    CONST robtarget Target_7240:=[[97.404735669,131.379041523,0],[0,0,1,0],[0,0,0,0],[9E+09,9E+09,9E+09,9E+09,9E+09,9E+09]];
    CONST robtarget Target_7250:=[[104.308059394,134.057322127,0],[0,0,1,0],[0,0,0,0],[9E+09,9E+09,9E+09,9E+09,9E+09,9E+09]];
    CONST robtarget Target_7260:=[[111.293699053,136.477383043,0],[0,0,1,0],[0,0,0,0],[9E+09,9E+09,9E+09,9E+09,9E+09,9E+09]];
    CONST robtarget Target_7270:=[[115.08379892,137.360119805,0],[0,0,1,0],[0,0,0,0],[9E+09,9E+09,9E+09,9E+09,9E+09,9E+09]];
    CONST robtarget Target_7280:=[[119.016514302,137.798137565,0],[0,0,1,0],[0,0,0,0],[9E+09,9E+09,9E+09,9E+09,9E+09,9E+09]];
    CONST robtarget Target_7290:=[[126.994438246,138.21544406,0],[0,0,1,0],[0,0,0,0],[9E+09,9E+09,9E+09,9E+09,9E+09,9E+09]];
    CONST robtarget Target_7300:=[[128.009308622,138.133836593,0],[0,0,1,0],[0,0,0,0],[9E+09,9E+09,9E+09,9E+09,9E+09,9E+09]];
    CONST robtarget Target_7310:=[[129.094775731,137.821862787,0],[0,0,1,0],[0,0,0,0],[9E+09,9E+09,9E+09,9E+09,9E+09,9E+09]];
    CONST robtarget Target_7320:=[[131.666016764,136.934701488,0],[0,0,1,0],[0,0,0,0],[9E+09,9E+09,9E+09,9E+09,9E+09,9E+09]];
    CONST robtarget Target_7330:=[[115.036980299,130.031874476,0],[0,0,1,0],[0,0,0,0],[9E+09,9E+09,9E+09,9E+09,9E+09,9E+09]];
    CONST robtarget Target_7330_2:=[[115.036980299,130.031874476,20],[0,0,1,0],[0,0,0,0],[9E+09,9E+09,9E+09,9E+09,9E+09,9E+09]];
    CONST robtarget Target_7340_2:=[[129.876572493,85.549987473,20],[0,0,1,0],[0,0,0,0],[9E+09,9E+09,9E+09,9E+09,9E+09,9E+09]];
    CONST robtarget Target_7340:=[[129.876572493,85.549987473,0],[0,0,1,0],[0,0,0,0],[9E+09,9E+09,9E+09,9E+09,9E+09,9E+09]];
    CONST robtarget Target_7350:=[[129.333218932,86.748318348,0],[0,0,1,0],[0,0,0,0],[9E+09,9E+09,9E+09,9E+09,9E+09,9E+09]];
    CONST robtarget Target_7360:=[[120.656332036,84.597871563,0],[0,0,1,0],[0,0,0,0],[9E+09,9E+09,9E+09,9E+09,9E+09,9E+09]];
    CONST robtarget Target_7370:=[[116.357422703,83.423068967,0],[0,0,1,0],[0,0,0,0],[9E+09,9E+09,9E+09,9E+09,9E+09,9E+09]];
    CONST robtarget Target_7380:=[[112.166530873,81.976192315,0],[0,0,1,0],[0,0,0,0],[9E+09,9E+09,9E+09,9E+09,9E+09,9E+09]];
    CONST robtarget Target_7390:=[[106.124575096,79.401977146,0],[0,0,1,0],[0,0,0,0],[9E+09,9E+09,9E+09,9E+09,9E+09,9E+09]];
    CONST robtarget Target_7400:=[[88.244330691,71.049330005,0],[0,0,1,0],[0,0,0,0],[9E+09,9E+09,9E+09,9E+09,9E+09,9E+09]];
    CONST robtarget Target_7410:=[[84.481212005,69.620753442,0],[0,0,1,0],[0,0,0,0],[9E+09,9E+09,9E+09,9E+09,9E+09,9E+09]];
    CONST robtarget Target_7420:=[[80.716429491,68.637006398,0],[0,0,1,0],[0,0,0,0],[9E+09,9E+09,9E+09,9E+09,9E+09,9E+09]];
    CONST robtarget Target_7430:=[[76.954340789,68.092878497,0],[0,0,1,0],[0,0,0,0],[9E+09,9E+09,9E+09,9E+09,9E+09,9E+09]];
    CONST robtarget Target_7440:=[[73.199303537,67.983159363,0],[0,0,1,0],[0,0,0,0],[9E+09,9E+09,9E+09,9E+09,9E+09,9E+09]];
    CONST robtarget Target_7450:=[[69.455675374,68.302638618,0],[0,0,1,0],[0,0,0,0],[9E+09,9E+09,9E+09,9E+09,9E+09,9E+09]];
    CONST robtarget Target_7460:=[[65.727813937,69.046105887,0],[0,0,1,0],[0,0,0,0],[9E+09,9E+09,9E+09,9E+09,9E+09,9E+09]];
    CONST robtarget Target_7470:=[[62.020076867,70.208350794,0],[0,0,1,0],[0,0,0,0],[9E+09,9E+09,9E+09,9E+09,9E+09,9E+09]];
    CONST robtarget Target_7480:=[[58.336821801,71.78416296,0],[0,0,1,0],[0,0,0,0],[9E+09,9E+09,9E+09,9E+09,9E+09,9E+09]];
    CONST robtarget Target_7490:=[[56.763326351,72.672328805,0],[0,0,1,0],[0,0,0,0],[9E+09,9E+09,9E+09,9E+09,9E+09,9E+09]];
    CONST robtarget Target_7500:=[[55.419669303,73.685478708,0],[0,0,1,0],[0,0,0,0],[9E+09,9E+09,9E+09,9E+09,9E+09,9E+09]];
    CONST robtarget Target_7510:=[[54.298199796,74.808495832,0],[0,0,1,0],[0,0,0,0],[9E+09,9E+09,9E+09,9E+09,9E+09,9E+09]];
    CONST robtarget Target_7520:=[[53.391266972,76.026263336,0],[0,0,1,0],[0,0,0,0],[9E+09,9E+09,9E+09,9E+09,9E+09,9E+09]];
    CONST robtarget Target_7530:=[[52.691219971,77.323664383,0],[0,0,1,0],[0,0,0,0],[9E+09,9E+09,9E+09,9E+09,9E+09,9E+09]];
    CONST robtarget Target_7540:=[[52.190407933,78.685582133,0],[0,0,1,0],[0,0,0,0],[9E+09,9E+09,9E+09,9E+09,9E+09,9E+09]];
    CONST robtarget Target_7550:=[[51.755885311,81.542500387,0],[0,0,1,0],[0,0,0,0],[9E+09,9E+09,9E+09,9E+09,9E+09,9E+09]];
    CONST robtarget Target_7560:=[[52.026492229,84.476083387,0],[0,0,1,0],[0,0,0,0],[9E+09,9E+09,9E+09,9E+09,9E+09,9E+09]];
    CONST robtarget Target_7570:=[[52.941021811,87.365396422,0],[0,0,1,0],[0,0,0,0],[9E+09,9E+09,9E+09,9E+09,9E+09,9E+09]];
    CONST robtarget Target_7580:=[[54.438267181,90.089504782,0],[0,0,1,0],[0,0,0,0],[9E+09,9E+09,9E+09,9E+09,9E+09,9E+09]];
    CONST robtarget Target_7590:=[[56.457021465,92.527473754,0],[0,0,1,0],[0,0,0,0],[9E+09,9E+09,9E+09,9E+09,9E+09,9E+09]];
    CONST robtarget Target_7600:=[[56.316335288,88.929115434,0],[0,0,1,0],[0,0,0,0],[9E+09,9E+09,9E+09,9E+09,9E+09,9E+09]];
    CONST robtarget Target_7610:=[[56.453523859,85.970317693,0],[0,0,1,0],[0,0,0,0],[9E+09,9E+09,9E+09,9E+09,9E+09,9E+09]];
    CONST robtarget Target_7620:=[[56.93899034,83.536042059,0],[0,0,1,0],[0,0,0,0],[9E+09,9E+09,9E+09,9E+09,9E+09,9E+09]];
    CONST robtarget Target_7630:=[[57.843137896,81.511250063,0],[0,0,1,0],[0,0,0,0],[9E+09,9E+09,9E+09,9E+09,9E+09,9E+09]];
    CONST robtarget Target_7640:=[[59.23636969,79.780903236,0],[0,0,1,0],[0,0,0,0],[9E+09,9E+09,9E+09,9E+09,9E+09,9E+09]];
    CONST robtarget Target_7650:=[[61.189088885,78.229963107,0],[0,0,1,0],[0,0,0,0],[9E+09,9E+09,9E+09,9E+09,9E+09,9E+09]];
    CONST robtarget Target_7660:=[[63.771698646,76.743391208,0],[0,0,1,0],[0,0,0,0],[9E+09,9E+09,9E+09,9E+09,9E+09,9E+09]];
    CONST robtarget Target_7670:=[[67.054602136,75.206149067,0],[0,0,1,0],[0,0,0,0],[9E+09,9E+09,9E+09,9E+09,9E+09,9E+09]];
    CONST robtarget Target_7680:=[[68.464100111,74.610784942,0],[0,0,1,0],[0,0,0,0],[9E+09,9E+09,9E+09,9E+09,9E+09,9E+09]];
    CONST robtarget Target_7690:=[[71.32349125,73.279802023,0],[0,0,1,0],[0,0,0,0],[9E+09,9E+09,9E+09,9E+09,9E+09,9E+09]];
    CONST robtarget Target_7700:=[[74.141087214,72.412520642,0],[0,0,1,0],[0,0,0,0],[9E+09,9E+09,9E+09,9E+09,9E+09,9E+09]];
    CONST robtarget Target_7710:=[[76.925445565,71.99176175,0],[0,0,1,0],[0,0,0,0],[9E+09,9E+09,9E+09,9E+09,9E+09,9E+09]];
    CONST robtarget Target_7720:=[[79.685123865,72.000346299,0],[0,0,1,0],[0,0,0,0],[9E+09,9E+09,9E+09,9E+09,9E+09,9E+09]];
    CONST robtarget Target_7730:=[[82.428679675,72.421095242,0],[0,0,1,0],[0,0,0,0],[9E+09,9E+09,9E+09,9E+09,9E+09,9E+09]];
    CONST robtarget Target_7740:=[[85.164670556,73.236829529,0],[0,0,1,0],[0,0,0,0],[9E+09,9E+09,9E+09,9E+09,9E+09,9E+09]];
    CONST robtarget Target_7750:=[[87.901654071,74.430370112,0],[0,0,1,0],[0,0,0,0],[9E+09,9E+09,9E+09,9E+09,9E+09,9E+09]];
    CONST robtarget Target_7760:=[[94.465610205,78.171040828,0],[0,0,1,0],[0,0,0,0],[9E+09,9E+09,9E+09,9E+09,9E+09,9E+09]];
    CONST robtarget Target_7770:=[[98.441342552,80.111743376,0],[0,0,1,0],[0,0,0,0],[9E+09,9E+09,9E+09,9E+09,9E+09,9E+09]];
    CONST robtarget Target_7780:=[[106.616652637,83.542913403,0],[0,0,1,0],[0,0,0,0],[9E+09,9E+09,9E+09,9E+09,9E+09,9E+09]];
    CONST robtarget Target_7790:=[[116.490797826,87.190723014,0],[0,0,1,0],[0,0,0,0],[9E+09,9E+09,9E+09,9E+09,9E+09,9E+09]];
    CONST robtarget Target_7800:=[[126.476326895,90.545417185,0],[0,0,1,0],[0,0,0,0],[9E+09,9E+09,9E+09,9E+09,9E+09,9E+09]];
    CONST robtarget Target_7810:=[[132.154721448,92.265104517,0],[0,0,1,0],[0,0,0,0],[9E+09,9E+09,9E+09,9E+09,9E+09,9E+09]];
    CONST robtarget Target_7820:=[[137.901994386,93.748799757,0],[0,0,1,0],[0,0,0,0],[9E+09,9E+09,9E+09,9E+09,9E+09,9E+09]];
    CONST robtarget Target_7830:=[[138.868681172,94.121198932,0],[0,0,1,0],[0,0,0,0],[9E+09,9E+09,9E+09,9E+09,9E+09,9E+09]];
    CONST robtarget Target_7840:=[[140.005403026,94.778288617,0],[0,0,1,0],[0,0,0,0],[9E+09,9E+09,9E+09,9E+09,9E+09,9E+09]];
    CONST robtarget Target_7850:=[[142.426589149,96.658715467,0],[0,0,1,0],[0,0,0,0],[9E+09,9E+09,9E+09,9E+09,9E+09,9E+09]];
    CONST robtarget Target_7860:=[[144.440827175,98.81443219,0],[0,0,1,0],[0,0,0,0],[9E+09,9E+09,9E+09,9E+09,9E+09,9E+09]];
    CONST robtarget Target_7870:=[[145.068863909,99.81563422,0],[0,0,1,0],[0,0,0,0],[9E+09,9E+09,9E+09,9E+09,9E+09,9E+09]];
    CONST robtarget Target_7880:=[[146.276657484,118.119049392,0],[0,0,1,0],[0,0,0,0],[9E+09,9E+09,9E+09,9E+09,9E+09,9E+09]];
    CONST robtarget Target_7890:=[[146.64526605,126.844242033,0],[0,0,1,0],[0,0,0,0],[9E+09,9E+09,9E+09,9E+09,9E+09,9E+09]];
    CONST robtarget Target_7900:=[[146.787973419,135.569206509,0],[0,0,1,0],[0,0,0,0],[9E+09,9E+09,9E+09,9E+09,9E+09,9E+09]];
    CONST robtarget Target_7910:=[[146.562475324,139.254038779,0],[0,0,1,0],[0,0,0,0],[9E+09,9E+09,9E+09,9E+09,9E+09,9E+09]];
    CONST robtarget Target_7920:=[[145.921246168,142.96350994,0],[0,0,1,0],[0,0,0,0],[9E+09,9E+09,9E+09,9E+09,9E+09,9E+09]];
    CONST robtarget Target_7930:=[[144.906271256,146.595460317,0],[0,0,1,0],[0,0,0,0],[9E+09,9E+09,9E+09,9E+09,9E+09,9E+09]];
    CONST robtarget Target_7940:=[[143.559535893,150.04773023,0],[0,0,1,0],[0,0,0,0],[9E+09,9E+09,9E+09,9E+09,9E+09,9E+09]];
    CONST robtarget Target_7950:=[[142.098362485,152.988920359,0],[0,0,1,0],[0,0,0,0],[9E+09,9E+09,9E+09,9E+09,9E+09,9E+09]];
    CONST robtarget Target_7960:=[[140.597343597,155.290040678,0],[0,0,1,0],[0,0,0,0],[9E+09,9E+09,9E+09,9E+09,9E+09,9E+09]];
    CONST robtarget Target_7970:=[[138.979884765,156.940428018,0],[0,0,1,0],[0,0,0,0],[9E+09,9E+09,9E+09,9E+09,9E+09,9E+09]];
    CONST robtarget Target_7980:=[[137.169391522,157.929419214,0],[0,0,1,0],[0,0,0,0],[9E+09,9E+09,9E+09,9E+09,9E+09,9E+09]];
    CONST robtarget Target_7990:=[[135.089269401,158.246351098,0],[0,0,1,0],[0,0,0,0],[9E+09,9E+09,9E+09,9E+09,9E+09,9E+09]];
    CONST robtarget Target_8000:=[[132.662923938,157.880560503,0],[0,0,1,0],[0,0,0,0],[9E+09,9E+09,9E+09,9E+09,9E+09,9E+09]];
    CONST robtarget Target_8010:=[[131.295981682,157.438312036,0],[0,0,1,0],[0,0,0,0],[9E+09,9E+09,9E+09,9E+09,9E+09,9E+09]];
    CONST robtarget Target_8020:=[[129.813760666,156.821384262,0],[0,0,1,0],[0,0,0,0],[9E+09,9E+09,9E+09,9E+09,9E+09,9E+09]];
    CONST robtarget Target_8030:=[[128.206686581,156.028444284,0],[0,0,1,0],[0,0,0,0],[9E+09,9E+09,9E+09,9E+09,9E+09,9E+09]];
    CONST robtarget Target_8040:=[[126.465185118,155.058159208,0],[0,0,1,0],[0,0,0,0],[9E+09,9E+09,9E+09,9E+09,9E+09,9E+09]];
    CONST robtarget Target_8050:=[[109.498646442,144.635036292,0],[0,0,1,0],[0,0,0,0],[9E+09,9E+09,9E+09,9E+09,9E+09,9E+09]];
    CONST robtarget Target_8060:=[[106.871095834,143.600815978,0],[0,0,1,0],[0,0,0,0],[9E+09,9E+09,9E+09,9E+09,9E+09,9E+09]];
    CONST robtarget Target_8070:=[[104.040074599,143.129604341,0],[0,0,1,0],[0,0,0,0],[9E+09,9E+09,9E+09,9E+09,9E+09,9E+09]];
    CONST robtarget Target_8080:=[[102.705166463,143.724153708,0],[0,0,1,0],[0,0,0,0],[9E+09,9E+09,9E+09,9E+09,9E+09,9E+09]];
    CONST robtarget Target_8090:=[[101.793162077,144.941800307,0],[0,0,1,0],[0,0,0,0],[9E+09,9E+09,9E+09,9E+09,9E+09,9E+09]];
    CONST robtarget Target_8100:=[[101.495618729,147.367025782,0],[0,0,1,0],[0,0,0,0],[9E+09,9E+09,9E+09,9E+09,9E+09,9E+09]];
    CONST robtarget Target_8110:=[[101.657829955,149.725149825,0],[0,0,1,0],[0,0,0,0],[9E+09,9E+09,9E+09,9E+09,9E+09,9E+09]];
    CONST robtarget Target_8120:=[[102.392934157,151.976800956,0],[0,0,1,0],[0,0,0,0],[9E+09,9E+09,9E+09,9E+09,9E+09,9E+09]];
    CONST robtarget Target_8130:=[[103.814069741,154.082607694,0],[0,0,1,0],[0,0,0,0],[9E+09,9E+09,9E+09,9E+09,9E+09,9E+09]];
    CONST robtarget Target_8140:=[[105.014427772,152.941872808,0],[0,0,1,0],[0,0,0,0],[9E+09,9E+09,9E+09,9E+09,9E+09,9E+09]];
    CONST robtarget Target_8150:=[[106.090948335,152.075840773,0],[0,0,1,0],[0,0,0,0],[9E+09,9E+09,9E+09,9E+09,9E+09,9E+09]];
    CONST robtarget Target_8160:=[[107.094496065,151.472364639,0],[0,0,1,0],[0,0,0,0],[9E+09,9E+09,9E+09,9E+09,9E+09,9E+09]];
    CONST robtarget Target_8170:=[[108.075935597,151.11929746,0],[0,0,1,0],[0,0,0,0],[9E+09,9E+09,9E+09,9E+09,9E+09,9E+09]];
    CONST robtarget Target_8180:=[[109.086131569,151.004492288,0],[0,0,1,0],[0,0,0,0],[9E+09,9E+09,9E+09,9E+09,9E+09,9E+09]];
    CONST robtarget Target_8190:=[[110.175948615,151.115802173,0],[0,0,1,0],[0,0,0,0],[9E+09,9E+09,9E+09,9E+09,9E+09,9E+09]];
    CONST robtarget Target_8200:=[[111.396251371,151.441080169,0],[0,0,1,0],[0,0,0,0],[9E+09,9E+09,9E+09,9E+09,9E+09,9E+09]];
    CONST robtarget Target_8210:=[[112.797904472,151.968179326,0],[0,0,1,0],[0,0,0,0],[9E+09,9E+09,9E+09,9E+09,9E+09,9E+09]];
    CONST robtarget Target_8220:=[[115.564679196,153.274276463,0],[0,0,1,0],[0,0,0,0],[9E+09,9E+09,9E+09,9E+09,9E+09,9E+09]];
    CONST robtarget Target_8230:=[[132.009061776,159.756169017,0],[0,0,1,0],[0,0,0,0],[9E+09,9E+09,9E+09,9E+09,9E+09,9E+09]];
    CONST robtarget Target_8240:=[[134.035319183,160.214476419,0],[0,0,1,0],[0,0,0,0],[9E+09,9E+09,9E+09,9E+09,9E+09,9E+09]];
    CONST robtarget Target_8250:=[[135.93027141,160.027374554,0],[0,0,1,0],[0,0,0,0],[9E+09,9E+09,9E+09,9E+09,9E+09,9E+09]];
    CONST robtarget Target_8260:=[[137.707220601,159.295275159,0],[0,0,1,0],[0,0,0,0],[9E+09,9E+09,9E+09,9E+09,9E+09,9E+09]];
    CONST robtarget Target_8270:=[[139.379468904,158.118589974,0],[0,0,1,0],[0,0,0,0],[9E+09,9E+09,9E+09,9E+09,9E+09,9E+09]];
    CONST robtarget Target_8280:=[[142.735905784,155.157330385,0],[0,0,1,0],[0,0,0,0],[9E+09,9E+09,9E+09,9E+09,9E+09,9E+09]];
    CONST robtarget Target_8290:=[[146.248814226,158.507504441,0],[0,0,1,0],[0,0,0,0],[9E+09,9E+09,9E+09,9E+09,9E+09,9E+09]];
    CONST robtarget Target_8300:=[[149.181567375,162.145043518,0],[0,0,1,0],[0,0,0,0],[9E+09,9E+09,9E+09,9E+09,9E+09,9E+09]];
    CONST robtarget Target_8310:=[[151.588027369,166.046590479,0],[0,0,1,0],[0,0,0,0],[9E+09,9E+09,9E+09,9E+09,9E+09,9E+09]];
    CONST robtarget Target_8320:=[[153.522056348,170.188788191,0],[0,0,1,0],[0,0,0,0],[9E+09,9E+09,9E+09,9E+09,9E+09,9E+09]];
    CONST robtarget Target_8330:=[[155.037516447,174.548279518,0],[0,0,1,0],[0,0,0,0],[9E+09,9E+09,9E+09,9E+09,9E+09,9E+09]];
    CONST robtarget Target_8340:=[[156.188269805,179.101707326,0],[0,0,1,0],[0,0,0,0],[9E+09,9E+09,9E+09,9E+09,9E+09,9E+09]];
    CONST robtarget Target_8350:=[[157.02817856,183.82571448,0],[0,0,1,0],[0,0,0,0],[9E+09,9E+09,9E+09,9E+09,9E+09,9E+09]];
    CONST robtarget Target_8360:=[[157.61110485,188.696943846,0],[0,0,1,0],[0,0,0,0],[9E+09,9E+09,9E+09,9E+09,9E+09,9E+09]];
    CONST robtarget Target_8370:=[[159.511653012,185.615301707,0],[0,0,1,0],[0,0,0,0],[9E+09,9E+09,9E+09,9E+09,9E+09,9E+09]];
    CONST robtarget Target_8380:=[[160.122702203,184.061896932,0],[0,0,1,0],[0,0,0,0],[9E+09,9E+09,9E+09,9E+09,9E+09,9E+09]];
    CONST robtarget Target_8390:=[[160.269289382,182.540597159,0],[0,0,1,0],[0,0,0,0],[9E+09,9E+09,9E+09,9E+09,9E+09,9E+09]];
    CONST robtarget Target_8400:=[[159.048038496,172.743082596,0],[0,0,1,0],[0,0,0,0],[9E+09,9E+09,9E+09,9E+09,9E+09,9E+09]];
    CONST robtarget Target_8410:=[[157.272759984,163.030465722,0],[0,0,1,0],[0,0,0,0],[9E+09,9E+09,9E+09,9E+09,9E+09,9E+09]];
    CONST robtarget Target_8420:=[[152.804879363,147.17888185,0],[0,0,1,0],[0,0,0,0],[9E+09,9E+09,9E+09,9E+09,9E+09,9E+09]];
    CONST robtarget Target_8430:=[[152.522164651,144.959220559,0],[0,0,1,0],[0,0,0,0],[9E+09,9E+09,9E+09,9E+09,9E+09,9E+09]];
    CONST robtarget Target_8440:=[[152.513150484,142.629190929,0],[0,0,1,0],[0,0,0,0],[9E+09,9E+09,9E+09,9E+09,9E+09,9E+09]];
    CONST robtarget Target_8450:=[[152.692927912,137.569820222,0],[0,0,1,0],[0,0,0,0],[9E+09,9E+09,9E+09,9E+09,9E+09,9E+09]];
    CONST robtarget Target_8460:=[[156.030442498,141.602150995,0],[0,0,1,0],[0,0,0,0],[9E+09,9E+09,9E+09,9E+09,9E+09,9E+09]];
    CONST robtarget Target_8470:=[[156.030442498,132.222722326,0],[0,0,1,0],[0,0,0,0],[9E+09,9E+09,9E+09,9E+09,9E+09,9E+09]];
    CONST robtarget Target_8480:=[[157.683142524,134.267528632,0],[0,0,1,0],[0,0,0,0],[9E+09,9E+09,9E+09,9E+09,9E+09,9E+09]];
    CONST robtarget Target_8490:=[[158.819369695,133.854983277,0],[0,0,1,0],[0,0,0,0],[9E+09,9E+09,9E+09,9E+09,9E+09,9E+09]];
    CONST robtarget Target_8500:=[[162.027841116,110.98600871,0],[0,0,1,0],[0,0,0,0],[9E+09,9E+09,9E+09,9E+09,9E+09,9E+09]];
    CONST robtarget Target_8510:=[[181.059601621,117.520426784,0],[0,0,1,0],[0,0,0,0],[9E+09,9E+09,9E+09,9E+09,9E+09,9E+09]];
    CONST robtarget Target_8520:=[[182.051540866,118.158620642,0],[0,0,1,0],[0,0,0,0],[9E+09,9E+09,9E+09,9E+09,9E+09,9E+09]];
    CONST robtarget Target_8530:=[[182.911149594,119.054153231,0],[0,0,1,0],[0,0,0,0],[9E+09,9E+09,9E+09,9E+09,9E+09,9E+09]];
    CONST robtarget Target_8540:=[[185.369337847,121.989158564,0],[0,0,1,0],[0,0,0,0],[9E+09,9E+09,9E+09,9E+09,9E+09,9E+09]];
    CONST robtarget Target_8550:=[[187.52283735,125.030421014,0],[0,0,1,0],[0,0,0,0],[9E+09,9E+09,9E+09,9E+09,9E+09,9E+09]];
    CONST robtarget Target_8560:=[[189.341962726,128.188894081,0],[0,0,1,0],[0,0,0,0],[9E+09,9E+09,9E+09,9E+09,9E+09,9E+09]];
    CONST robtarget Target_8570:=[[190.797028597,131.475531266,0],[0,0,1,0],[0,0,0,0],[9E+09,9E+09,9E+09,9E+09,9E+09,9E+09]];
    CONST robtarget Target_8580:=[[191.858349584,134.90128607,0],[0,0,1,0],[0,0,0,0],[9E+09,9E+09,9E+09,9E+09,9E+09,9E+09]];
    CONST robtarget Target_8590:=[[192.496240311,138.477111994,0],[0,0,1,0],[0,0,0,0],[9E+09,9E+09,9E+09,9E+09,9E+09,9E+09]];
    CONST robtarget Target_8600:=[[192.6810154,142.213962539,0],[0,0,1,0],[0,0,0,0],[9E+09,9E+09,9E+09,9E+09,9E+09,9E+09]];
    CONST robtarget Target_8610:=[[192.382989472,146.122791206,0],[0,0,1,0],[0,0,0,0],[9E+09,9E+09,9E+09,9E+09,9E+09,9E+09]];
    CONST robtarget Target_8620:=[[192.420926442,148.208812875,0],[0,0,1,0],[0,0,0,0],[9E+09,9E+09,9E+09,9E+09,9E+09,9E+09]];
    CONST robtarget Target_8630:=[[192.684959714,150.325900139,0],[0,0,1,0],[0,0,0,0],[9E+09,9E+09,9E+09,9E+09,9E+09,9E+09]];
    CONST robtarget Target_8640:=[[194.072232654,150.218826726,0],[0,0,1,0],[0,0,0,0],[9E+09,9E+09,9E+09,9E+09,9E+09,9E+09]];
    CONST robtarget Target_8650:=[[195.747139356,143.338811976,0],[0,0,1,0],[0,0,0,0],[9E+09,9E+09,9E+09,9E+09,9E+09,9E+09]];
    CONST robtarget Target_8660:=[[196.664125368,136.503126165,0],[0,0,1,0],[0,0,0,0],[9E+09,9E+09,9E+09,9E+09,9E+09,9E+09]];
    CONST robtarget Target_8670:=[[196.884999904,129.708154654,0],[0,0,1,0],[0,0,0,0],[9E+09,9E+09,9E+09,9E+09,9E+09,9E+09]];
    CONST robtarget Target_8680:=[[196.471572174,122.950282803,0],[0,0,1,0],[0,0,0,0],[9E+09,9E+09,9E+09,9E+09,9E+09,9E+09]];
    CONST robtarget Target_8690:=[[195.485651391,116.22589597,0],[0,0,1,0],[0,0,0,0],[9E+09,9E+09,9E+09,9E+09,9E+09,9E+09]];
    CONST robtarget Target_8700:=[[193.989046766,109.531379516,0],[0,0,1,0],[0,0,0,0],[9E+09,9E+09,9E+09,9E+09,9E+09,9E+09]];
    CONST robtarget Target_8710:=[[192.043567513,102.863118799,0],[0,0,1,0],[0,0,0,0],[9E+09,9E+09,9E+09,9E+09,9E+09,9E+09]];
    CONST robtarget Target_8720:=[[189.711022843,96.217499179,0],[0,0,1,0],[0,0,0,0],[9E+09,9E+09,9E+09,9E+09,9E+09,9E+09]];
    CONST robtarget Target_8730:=[[196.507207134,106.638206483,0],[0,0,1,0],[0,0,0,0],[9E+09,9E+09,9E+09,9E+09,9E+09,9E+09]];
    CONST robtarget Target_8740:=[[194.822794884,94.14058975,0],[0,0,1,0],[0,0,0,0],[9E+09,9E+09,9E+09,9E+09,9E+09,9E+09]];
    CONST robtarget Target_8750:=[[191.767984454,82.136505163,0],[0,0,1,0],[0,0,0,0],[9E+09,9E+09,9E+09,9E+09,9E+09,9E+09]];
    CONST robtarget Target_8760:=[[188.283605859,70.215200936,0],[0,0,1,0],[0,0,0,0],[9E+09,9E+09,9E+09,9E+09,9E+09,9E+09]];
    CONST robtarget Target_8770:=[[184.439576675,58.342610969,0],[0,0,1,0],[0,0,0,0],[9E+09,9E+09,9E+09,9E+09,9E+09,9E+09]];
    CONST robtarget Target_8780:=[[191.596791989,64.817986988,0],[0,0,1,0],[0,0,0,0],[9E+09,9E+09,9E+09,9E+09,9E+09,9E+09]];
    CONST robtarget Target_8790:=[[192.600244759,63.94724308,0],[0,0,1,0],[0,0,0,0],[9E+09,9E+09,9E+09,9E+09,9E+09,9E+09]];
    CONST robtarget Target_8800:=[[181.316386808,45.55735645,0],[0,0,1,0],[0,0,0,0],[9E+09,9E+09,9E+09,9E+09,9E+09,9E+09]];
    CONST robtarget Target_8810:=[[180.372261691,43.421039482,0],[0,0,1,0],[0,0,0,0],[9E+09,9E+09,9E+09,9E+09,9E+09,9E+09]];
    CONST robtarget Target_8820:=[[180.129144821,42.280955318,0],[0,0,1,0],[0,0,0,0],[9E+09,9E+09,9E+09,9E+09,9E+09,9E+09]];
    CONST robtarget Target_8830:=[[180.119797422,41.18562281,0],[0,0,1,0],[0,0,0,0],[9E+09,9E+09,9E+09,9E+09,9E+09,9E+09]];
    CONST robtarget Target_8840:=[[180.601400728,38.257669681,0],[0,0,1,0],[0,0,0,0],[9E+09,9E+09,9E+09,9E+09,9E+09,9E+09]];
    CONST robtarget Target_8850:=[[181.314808838,35.434360847,0],[0,0,1,0],[0,0,0,0],[9E+09,9E+09,9E+09,9E+09,9E+09,9E+09]];
    CONST robtarget Target_8860:=[[182.251851673,32.713303093,0],[0,0,1,0],[0,0,0,0],[9E+09,9E+09,9E+09,9E+09,9E+09,9E+09]];
    CONST robtarget Target_8870:=[[183.404359151,30.092103202,0],[0,0,1,0],[0,0,0,0],[9E+09,9E+09,9E+09,9E+09,9E+09,9E+09]];
    CONST robtarget Target_8880:=[[184.764161193,27.56836796,0],[0,0,1,0],[0,0,0,0],[9E+09,9E+09,9E+09,9E+09,9E+09,9E+09]];
    CONST robtarget Target_8890:=[[186.323087717,25.13970415,0],[0,0,1,0],[0,0,0,0],[9E+09,9E+09,9E+09,9E+09,9E+09,9E+09]];
    CONST robtarget Target_8900:=[[188.072968645,22.803718557,0],[0,0,1,0],[0,0,0,0],[9E+09,9E+09,9E+09,9E+09,9E+09,9E+09]];
    CONST robtarget Target_8910:=[[190.005633895,20.558017965,0],[0,0,1,0],[0,0,0,0],[9E+09,9E+09,9E+09,9E+09,9E+09,9E+09]];
    CONST robtarget Target_8920:=[[192.020885573,18.577072276,0],[0,0,1,0],[0,0,0,0],[9E+09,9E+09,9E+09,9E+09,9E+09,9E+09]];
    CONST robtarget Target_8930:=[[194.22441566,16.936248541,0],[0,0,1,0],[0,0,0,0],[9E+09,9E+09,9E+09,9E+09,9E+09,9E+09]];
    CONST robtarget Target_8940:=[[196.702778083,15.717678967,0],[0,0,1,0],[0,0,0,0],[9E+09,9E+09,9E+09,9E+09,9E+09,9E+09]];
    CONST robtarget Target_8950:=[[199.542526769,15.003495761,0],[0,0,1,0],[0,0,0,0],[9E+09,9E+09,9E+09,9E+09,9E+09,9E+09]];
    CONST robtarget Target_8960:=[[201.153882275,14.877956022,0],[0,0,1,0],[0,0,0,0],[9E+09,9E+09,9E+09,9E+09,9E+09,9E+09]];
    CONST robtarget Target_8970:=[[202.564135721,14.991268303,0],[0,0,1,0],[0,0,0,0],[9E+09,9E+09,9E+09,9E+09,9E+09,9E+09]];
    CONST robtarget Target_8980:=[[203.767899383,15.347108916,0],[0,0,1,0],[0,0,0,0],[9E+09,9E+09,9E+09,9E+09,9E+09,9E+09]];
    CONST robtarget Target_8990:=[[204.759785534,15.949154177,0],[0,0,1,0],[0,0,0,0],[9E+09,9E+09,9E+09,9E+09,9E+09,9E+09]];
    CONST robtarget Target_9000:=[[205.534406448,16.801080396,0],[0,0,1,0],[0,0,0,0],[9E+09,9E+09,9E+09,9E+09,9E+09,9E+09]];
    CONST robtarget Target_9010:=[[206.086374398,17.906563889,0],[0,0,1,0],[0,0,0,0],[9E+09,9E+09,9E+09,9E+09,9E+09,9E+09]];
    CONST robtarget Target_9020:=[[206.41030166,19.269280967,0],[0,0,1,0],[0,0,0,0],[9E+09,9E+09,9E+09,9E+09,9E+09,9E+09]];
    CONST robtarget Target_9030:=[[206.500800507,20.892907944,0],[0,0,1,0],[0,0,0,0],[9E+09,9E+09,9E+09,9E+09,9E+09,9E+09]];
    CONST robtarget Target_9040:=[[206.185218881,23.076640763,0],[0,0,1,0],[0,0,0,0],[9E+09,9E+09,9E+09,9E+09,9E+09,9E+09]];
    CONST robtarget Target_9050:=[[205.382591695,24.995387031,0],[0,0,1,0],[0,0,0,0],[9E+09,9E+09,9E+09,9E+09,9E+09,9E+09]];
    CONST robtarget Target_9060:=[[204.197106581,26.718523927,0],[0,0,1,0],[0,0,0,0],[9E+09,9E+09,9E+09,9E+09,9E+09,9E+09]];
    CONST robtarget Target_9070:=[[202.732951174,28.315428627,0],[0,0,1,0],[0,0,0,0],[9E+09,9E+09,9E+09,9E+09,9E+09,9E+09]];
    CONST robtarget Target_9080:=[[201.23516049,29.821989131,0],[0,0,1,0],[0,0,0,0],[9E+09,9E+09,9E+09,9E+09,9E+09,9E+09]];
    CONST robtarget Target_9090:=[[199.891820974,31.444879405,0],[0,0,1,0],[0,0,0,0],[9E+09,9E+09,9E+09,9E+09,9E+09,9E+09]];
    CONST robtarget Target_9100:=[[198.917384536,33.31544624,0],[0,0,1,0],[0,0,0,0],[9E+09,9E+09,9E+09,9E+09,9E+09,9E+09]];
    CONST robtarget Target_9110:=[[198.635521194,34.384654239,0],[0,0,1,0],[0,0,0,0],[9E+09,9E+09,9E+09,9E+09,9E+09,9E+09]];
    CONST robtarget Target_9120:=[[198.526303089,35.565036423,0],[0,0,1,0],[0,0,0,0],[9E+09,9E+09,9E+09,9E+09,9E+09,9E+09]];
    CONST robtarget Target_9130:=[[200.025047194,34.332688531,0],[0,0,1,0],[0,0,0,0],[9E+09,9E+09,9E+09,9E+09,9E+09,9E+09]];
    CONST robtarget Target_9140:=[[201.408478298,33.350226146,0],[0,0,1,0],[0,0,0,0],[9E+09,9E+09,9E+09,9E+09,9E+09,9E+09]];
    CONST robtarget Target_9150:=[[202.710907397,32.605760367,0],[0,0,1,0],[0,0,0,0],[9E+09,9E+09,9E+09,9E+09,9E+09,9E+09]];
    CONST robtarget Target_9160:=[[203.966645486,32.08740229,0],[0,0,1,0],[0,0,0,0],[9E+09,9E+09,9E+09,9E+09,9E+09,9E+09]];
    CONST robtarget Target_9170:=[[205.210003564,31.783263015,0],[0,0,1,0],[0,0,0,0],[9E+09,9E+09,9E+09,9E+09,9E+09,9E+09]];
    CONST robtarget Target_9180:=[[206.475292626,31.681453639,0],[0,0,1,0],[0,0,0,0],[9E+09,9E+09,9E+09,9E+09,9E+09,9E+09]];
    CONST robtarget Target_9190:=[[207.796823668,31.77008526,0],[0,0,1,0],[0,0,0,0],[9E+09,9E+09,9E+09,9E+09,9E+09,9E+09]];
    CONST robtarget Target_9200:=[[209.208907689,32.037268976,0],[0,0,1,0],[0,0,0,0],[9E+09,9E+09,9E+09,9E+09,9E+09,9E+09]];
    CONST robtarget Target_9210:=[[206.498192883,34.63263406,0],[0,0,1,0],[0,0,0,0],[9E+09,9E+09,9E+09,9E+09,9E+09,9E+09]];
    CONST robtarget Target_9220:=[[204.288706623,36.849937851,0],[0,0,1,0],[0,0,0,0],[9E+09,9E+09,9E+09,9E+09,9E+09,9E+09]];
    CONST robtarget Target_9230:=[[202.519543794,38.803163097,0],[0,0,1,0],[0,0,0,0],[9E+09,9E+09,9E+09,9E+09,9E+09,9E+09]];
    CONST robtarget Target_9240:=[[201.129799285,40.606292545,0],[0,0,1,0],[0,0,0,0],[9E+09,9E+09,9E+09,9E+09,9E+09,9E+09]];
    CONST robtarget Target_9250:=[[200.058567982,42.373308942,0],[0,0,1,0],[0,0,0,0],[9E+09,9E+09,9E+09,9E+09,9E+09,9E+09]];
    CONST robtarget Target_9260:=[[199.244944772,44.218195037,0],[0,0,1,0],[0,0,0,0],[9E+09,9E+09,9E+09,9E+09,9E+09,9E+09]];
    CONST robtarget Target_9270:=[[198.628024542,46.254933577,0],[0,0,1,0],[0,0,0,0],[9E+09,9E+09,9E+09,9E+09,9E+09,9E+09]];
    CONST robtarget Target_9280:=[[198.146902179,48.597507309,0],[0,0,1,0],[0,0,0,0],[9E+09,9E+09,9E+09,9E+09,9E+09,9E+09]];
    CONST robtarget Target_9290:=[[196.61288422,59.686081257,0],[0,0,1,0],[0,0,0,0],[9E+09,9E+09,9E+09,9E+09,9E+09,9E+09]];
    CONST robtarget Target_9300:=[[196.174396262,65.230484615,0],[0,0,1,0],[0,0,0,0],[9E+09,9E+09,9E+09,9E+09,9E+09,9E+09]];
    CONST robtarget Target_9310:=[[196.004662814,70.774974464,0],[0,0,1,0],[0,0,0,0],[9E+09,9E+09,9E+09,9E+09,9E+09,9E+09]];
    CONST robtarget Target_9320:=[[196.140989249,76.31955748,0],[0,0,1,0],[0,0,0,0],[9E+09,9E+09,9E+09,9E+09,9E+09,9E+09]];
    CONST robtarget Target_9330:=[[196.620680938,81.864240338,0],[0,0,1,0],[0,0,0,0],[9E+09,9E+09,9E+09,9E+09,9E+09,9E+09]];
    CONST robtarget Target_9340:=[[197.481043255,87.409029715,0],[0,0,1,0],[0,0,0,0],[9E+09,9E+09,9E+09,9E+09,9E+09,9E+09]];
    CONST robtarget Target_9350:=[[198.759381571,92.953932286,0],[0,0,1,0],[0,0,0,0],[9E+09,9E+09,9E+09,9E+09,9E+09,9E+09]];
    CONST robtarget Target_9360:=[[201.564466199,104.252177175,0],[0,0,1,0],[0,0,0,0],[9E+09,9E+09,9E+09,9E+09,9E+09,9E+09]];
    CONST robtarget Target_9370:=[[203.789655734,115.652677805,0],[0,0,1,0],[0,0,0,0],[9E+09,9E+09,9E+09,9E+09,9E+09,9E+09]];
    CONST robtarget Target_9380:=[[204.636408963,121.396078998,0],[0,0,1,0],[0,0,0,0],[9E+09,9E+09,9E+09,9E+09,9E+09,9E+09]];
    CONST robtarget Target_9390:=[[205.280131364,127.170810095,0],[0,0,1,0],[0,0,0,0],[9E+09,9E+09,9E+09,9E+09,9E+09,9E+09]];
    CONST robtarget Target_9400:=[[205.701470586,132.978793087,0],[0,0,1,0],[0,0,0,0],[9E+09,9E+09,9E+09,9E+09,9E+09,9E+09]];
    CONST robtarget Target_9410:=[[205.881074278,138.821949962,0],[0,0,1,0],[0,0,0,0],[9E+09,9E+09,9E+09,9E+09,9E+09,9E+09]];
    CONST robtarget Target_9420:=[[205.923787544,163.023012903,0],[0,0,1,0],[0,0,0,0],[9E+09,9E+09,9E+09,9E+09,9E+09,9E+09]];
    CONST robtarget Target_9430:=[[206.224124409,164.437566789,0],[0,0,1,0],[0,0,0,0],[9E+09,9E+09,9E+09,9E+09,9E+09,9E+09]];
    CONST robtarget Target_9440:=[[206.729796792,165.850533718,0],[0,0,1,0],[0,0,0,0],[9E+09,9E+09,9E+09,9E+09,9E+09,9E+09]];
    CONST robtarget Target_9450:=[[207.958631791,165.588804952,0],[0,0,1,0],[0,0,0,0],[9E+09,9E+09,9E+09,9E+09,9E+09,9E+09]];
    CONST robtarget Target_9460:=[[207.958631791,150.141115173,0],[0,0,1,0],[0,0,0,0],[9E+09,9E+09,9E+09,9E+09,9E+09,9E+09]];
    CONST robtarget Target_9470:=[[209.430226624,151.721456097,0],[0,0,1,0],[0,0,0,0],[9E+09,9E+09,9E+09,9E+09,9E+09,9E+09]];
    CONST robtarget Target_9480:=[[210.695447211,153.379474728,0],[0,0,1,0],[0,0,0,0],[9E+09,9E+09,9E+09,9E+09,9E+09,9E+09]];
    CONST robtarget Target_9490:=[[211.761289196,155.107679103,0],[0,0,1,0],[0,0,0,0],[9E+09,9E+09,9E+09,9E+09,9E+09,9E+09]];
    CONST robtarget Target_9500:=[[212.634748223,156.898577253,0],[0,0,1,0],[0,0,0,0],[9E+09,9E+09,9E+09,9E+09,9E+09,9E+09]];
    CONST robtarget Target_9510:=[[213.832499974,160.638487019,0],[0,0,1,0],[0,0,0,0],[9E+09,9E+09,9E+09,9E+09,9E+09,9E+09]];
    CONST robtarget Target_9520:=[[214.344667613,164.539268295,0],[0,0,1,0],[0,0,0,0],[9E+09,9E+09,9E+09,9E+09,9E+09,9E+09]];
    CONST robtarget Target_9530:=[[215.042181606,177.509334354,0],[0,0,1,0],[0,0,0,0],[9E+09,9E+09,9E+09,9E+09,9E+09,9E+09]];
    CONST robtarget Target_9540:=[[215.288779154,183.99202098,0],[0,0,1,0],[0,0,0,0],[9E+09,9E+09,9E+09,9E+09,9E+09,9E+09]];
    CONST robtarget Target_9550:=[[215.321559695,190.464065247,0],[0,0,1,0],[0,0,0,0],[9E+09,9E+09,9E+09,9E+09,9E+09,9E+09]];
    CONST robtarget Target_9560:=[[215.0312402,196.918658587,0],[0,0,1,0],[0,0,0,0],[9E+09,9E+09,9E+09,9E+09,9E+09,9E+09]];
    CONST robtarget Target_9570:=[[214.308537638,203.348992435,0],[0,0,1,0],[0,0,0,0],[9E+09,9E+09,9E+09,9E+09,9E+09,9E+09]];
    CONST robtarget Target_9580:=[[213.044168979,209.748258222,0],[0,0,1,0],[0,0,0,0],[9E+09,9E+09,9E+09,9E+09,9E+09,9E+09]];
    CONST robtarget Target_9590:=[[211.128851192,216.109647382,0],[0,0,1,0],[0,0,0,0],[9E+09,9E+09,9E+09,9E+09,9E+09,9E+09]];
    CONST robtarget Target_9600:=[[210.788553003,217.797412552,0],[0,0,1,0],[0,0,0,0],[9E+09,9E+09,9E+09,9E+09,9E+09,9E+09]];
    CONST robtarget Target_9610:=[[210.788455864,219.607370654,0],[0,0,1,0],[0,0,0,0],[9E+09,9E+09,9E+09,9E+09,9E+09,9E+09]];
    CONST robtarget Target_9620:=[[211.023875056,223.31191667,0],[0,0,1,0],[0,0,0,0],[9E+09,9E+09,9E+09,9E+09,9E+09,9E+09]];
    CONST robtarget Target_9630:=[[212.166253612,223.389478418,0],[0,0,1,0],[0,0,0,0],[9E+09,9E+09,9E+09,9E+09,9E+09,9E+09]];
    CONST robtarget Target_9640:=[[214.81517292,218.24211088,0],[0,0,1,0],[0,0,0,0],[9E+09,9E+09,9E+09,9E+09,9E+09,9E+09]];
    CONST robtarget Target_9650:=[[216.899235082,212.99446713,0],[0,0,1,0],[0,0,0,0],[9E+09,9E+09,9E+09,9E+09,9E+09,9E+09]];
    CONST robtarget Target_9660:=[[218.451485575,207.65318286,0],[0,0,1,0],[0,0,0,0],[9E+09,9E+09,9E+09,9E+09,9E+09,9E+09]];
    CONST robtarget Target_9670:=[[219.504969875,202.224893763,0],[0,0,1,0],[0,0,0,0],[9E+09,9E+09,9E+09,9E+09,9E+09,9E+09]];
    CONST robtarget Target_9680:=[[220.09273346,196.71623553,0],[0,0,1,0],[0,0,0,0],[9E+09,9E+09,9E+09,9E+09,9E+09,9E+09]];
    CONST robtarget Target_9690:=[[220.247821808,191.133843852,0],[0,0,1,0],[0,0,0,0],[9E+09,9E+09,9E+09,9E+09,9E+09,9E+09]];
    CONST robtarget Target_9700:=[[220.003280397,185.484354422,0],[0,0,1,0],[0,0,0,0],[9E+09,9E+09,9E+09,9E+09,9E+09,9E+09]];
    CONST robtarget Target_9710:=[[219.392154702,179.774402932,0],[0,0,1,0],[0,0,0,0],[9E+09,9E+09,9E+09,9E+09,9E+09,9E+09]];
    CONST robtarget Target_9720:=[[222.818953308,182.875955281,0],[0,0,1,0],[0,0,0,0],[9E+09,9E+09,9E+09,9E+09,9E+09,9E+09]];
    CONST robtarget Target_9730:=[[221.216466181,170.263445118,0],[0,0,1,0],[0,0,0,0],[9E+09,9E+09,9E+09,9E+09,9E+09,9E+09]];
    CONST robtarget Target_9740:=[[224.690584569,174.489773888,0],[0,0,1,0],[0,0,0,0],[9E+09,9E+09,9E+09,9E+09,9E+09,9E+09]];
    CONST robtarget Target_9750:=[[222.932224919,158.594053599,0],[0,0,1,0],[0,0,0,0],[9E+09,9E+09,9E+09,9E+09,9E+09,9E+09]];
    CONST robtarget Target_9760:=[[226.388937265,160.242686447,0],[0,0,1,0],[0,0,0,0],[9E+09,9E+09,9E+09,9E+09,9E+09,9E+09]];
    CONST robtarget Target_9770:=[[229.163511759,162.160527018,0],[0,0,1,0],[0,0,0,0],[9E+09,9E+09,9E+09,9E+09,9E+09,9E+09]];
    CONST robtarget Target_9780:=[[231.64146646,163.780277585,0],[0,0,1,0],[0,0,0,0],[9E+09,9E+09,9E+09,9E+09,9E+09,9E+09]];
    CONST robtarget Target_9790:=[[233.664364267,165.750085982,0],[0,0,1,0],[0,0,0,0],[9E+09,9E+09,9E+09,9E+09,9E+09,9E+09]];
    CONST robtarget Target_9800:=[[235.150974787,168.07083855,0],[0,0,1,0],[0,0,0,0],[9E+09,9E+09,9E+09,9E+09,9E+09,9E+09]];
    CONST robtarget Target_9810:=[[236.020067627,170.743421631,0],[0,0,1,0],[0,0,0,0],[9E+09,9E+09,9E+09,9E+09,9E+09,9E+09]];
    CONST robtarget Target_9820:=[[237.32517248,179.926984083,0],[0,0,1,0],[0,0,0,0],[9E+09,9E+09,9E+09,9E+09,9E+09,9E+09]];
    CONST robtarget Target_9830:=[[238.319449492,189.168231645,0],[0,0,1,0],[0,0,0,0],[9E+09,9E+09,9E+09,9E+09,9E+09,9E+09]];
    CONST robtarget Target_9840:=[[238.647148812,192.721166401,0],[0,0,1,0],[0,0,0,0],[9E+09,9E+09,9E+09,9E+09,9E+09,9E+09]];
    CONST robtarget Target_9850:=[[239.775582628,191.346305695,0],[0,0,1,0],[0,0,0,0],[9E+09,9E+09,9E+09,9E+09,9E+09,9E+09]];
    CONST robtarget Target_9860:=[[240.63708099,189.923062745,0],[0,0,1,0],[0,0,0,0],[9E+09,9E+09,9E+09,9E+09,9E+09,9E+09]];
    CONST robtarget Target_9870:=[[241.260450643,188.454150066,0],[0,0,1,0],[0,0,0,0],[9E+09,9E+09,9E+09,9E+09,9E+09,9E+09]];
    CONST robtarget Target_9880:=[[241.674498331,186.942280176,0],[0,0,1,0],[0,0,0,0],[9E+09,9E+09,9E+09,9E+09,9E+09,9E+09]];
    CONST robtarget Target_9890:=[[241.989854798,183.800518828,0],[0,0,1,0],[0,0,0,0],[9E+09,9E+09,9E+09,9E+09,9E+09,9E+09]];
    CONST robtarget Target_9900:=[[241.813604352,180.519478832,0],[0,0,1,0],[0,0,0,0],[9E+09,9E+09,9E+09,9E+09,9E+09,9E+09]];
    CONST robtarget Target_9910:=[[243.450961978,182.059334288,0],[0,0,1,0],[0,0,0,0],[9E+09,9E+09,9E+09,9E+09,9E+09,9E+09]];
    CONST robtarget Target_9920:=[[244.865637571,183.923582614,0],[0,0,1,0],[0,0,0,0],[9E+09,9E+09,9E+09,9E+09,9E+09,9E+09]];
    CONST robtarget Target_9930:=[[246.036209313,186.034041308,0],[0,0,1,0],[0,0,0,0],[9E+09,9E+09,9E+09,9E+09,9E+09,9E+09]];
    CONST robtarget Target_9940:=[[246.941255387,188.312527869,0],[0,0,1,0],[0,0,0,0],[9E+09,9E+09,9E+09,9E+09,9E+09,9E+09]];
    CONST robtarget Target_9950:=[[247.559353976,190.680859793,0],[0,0,1,0],[0,0,0,0],[9E+09,9E+09,9E+09,9E+09,9E+09,9E+09]];
    CONST robtarget Target_9960:=[[247.869083262,193.060854579,0],[0,0,1,0],[0,0,0,0],[9E+09,9E+09,9E+09,9E+09,9E+09,9E+09]];
    CONST robtarget Target_9970:=[[247.849021429,195.374329726,0],[0,0,1,0],[0,0,0,0],[9E+09,9E+09,9E+09,9E+09,9E+09,9E+09]];
    CONST robtarget Target_9980:=[[247.47774666,197.54310273,0],[0,0,1,0],[0,0,0,0],[9E+09,9E+09,9E+09,9E+09,9E+09,9E+09]];
    CONST robtarget Target_9990:=[[247.177218294,200.687536876,0],[0,0,1,0],[0,0,0,0],[9E+09,9E+09,9E+09,9E+09,9E+09,9E+09]];
    CONST robtarget Target_10000:=[[248.35852753,200.953141856,0],[0,0,1,0],[0,0,0,0],[9E+09,9E+09,9E+09,9E+09,9E+09,9E+09]];
    CONST robtarget Target_10010:=[[251.109198172,194.054621749,0],[0,0,1,0],[0,0,0,0],[9E+09,9E+09,9E+09,9E+09,9E+09,9E+09]];
    CONST robtarget Target_10020:=[[251.968576839,196.91465564,0],[0,0,1,0],[0,0,0,0],[9E+09,9E+09,9E+09,9E+09,9E+09,9E+09]];
    CONST robtarget Target_10030:=[[252.189721726,199.681527173,0],[0,0,1,0],[0,0,0,0],[9E+09,9E+09,9E+09,9E+09,9E+09,9E+09]];
    CONST robtarget Target_10040:=[[251.931642346,202.381817081,0],[0,0,1,0],[0,0,0,0],[9E+09,9E+09,9E+09,9E+09,9E+09,9E+09]];
    CONST robtarget Target_10050:=[[251.35334821,205.042106094,0],[0,0,1,0],[0,0,0,0],[9E+09,9E+09,9E+09,9E+09,9E+09,9E+09]];
    CONST robtarget Target_10060:=[[249.87215372,210.349004354,0],[0,0,1,0],[0,0,0,0],[9E+09,9E+09,9E+09,9E+09,9E+09,9E+09]];
    CONST robtarget Target_10070:=[[249.287272389,213.048775063,0],[0,0,1,0],[0,0,0,0],[9E+09,9E+09,9E+09,9E+09,9E+09,9E+09]];
    CONST robtarget Target_10080:=[[249.01821435,215.814867799,0],[0,0,1,0],[0,0,0,0],[9E+09,9E+09,9E+09,9E+09,9E+09,9E+09]];
    CONST robtarget Target_10090:=[[256.680760741,208.892809518,0],[0,0,1,0],[0,0,0,0],[9E+09,9E+09,9E+09,9E+09,9E+09,9E+09]];
    CONST robtarget Target_10100:=[[256.856099046,212.124809519,0],[0,0,1,0],[0,0,0,0],[9E+09,9E+09,9E+09,9E+09,9E+09,9E+09]];
    CONST robtarget Target_10110:=[[256.851499022,213.421939973,0],[0,0,1,0],[0,0,0,0],[9E+09,9E+09,9E+09,9E+09,9E+09,9E+09]];
    CONST robtarget Target_10120:=[[256.586476965,214.524893469,0],[0,0,1,0],[0,0,0,0],[9E+09,9E+09,9E+09,9E+09,9E+09,9E+09]];
    CONST robtarget Target_10130:=[[253.755293806,220.274941697,0],[0,0,1,0],[0,0,0,0],[9E+09,9E+09,9E+09,9E+09,9E+09,9E+09]];
    CONST robtarget Target_10140:=[[250.784832022,225.822514791,0],[0,0,1,0],[0,0,0,0],[9E+09,9E+09,9E+09,9E+09,9E+09,9E+09]];
    CONST robtarget Target_10150:=[[252.157252939,225.315949552,0],[0,0,1,0],[0,0,0,0],[9E+09,9E+09,9E+09,9E+09,9E+09,9E+09]];
    CONST robtarget Target_10160:=[[253.831162355,224.925873274,0],[0,0,1,0],[0,0,0,0],[9E+09,9E+09,9E+09,9E+09,9E+09,9E+09]];
    CONST robtarget Target_10170:=[[255.063434717,225.199761821,0],[0,0,1,0],[0,0,0,0],[9E+09,9E+09,9E+09,9E+09,9E+09,9E+09]];
    CONST robtarget Target_10180:=[[255.970027729,225.94462492,0],[0,0,1,0],[0,0,0,0],[9E+09,9E+09,9E+09,9E+09,9E+09,9E+09]];
    CONST robtarget Target_10190:=[[256.167629907,228.159069348,0],[0,0,1,0],[0,0,0,0],[9E+09,9E+09,9E+09,9E+09,9E+09,9E+09]];
    CONST robtarget Target_10200:=[[255.530555132,231.175044904,0],[0,0,1,0],[0,0,0,0],[9E+09,9E+09,9E+09,9E+09,9E+09,9E+09]];
    CONST robtarget Target_10210:=[[254.377007363,234.09268169,0],[0,0,1,0],[0,0,0,0],[9E+09,9E+09,9E+09,9E+09,9E+09,9E+09]];
    CONST robtarget Target_10220:=[[253.705994843,235.233413701,0],[0,0,1,0],[0,0,0,0],[9E+09,9E+09,9E+09,9E+09,9E+09,9E+09]];
    CONST robtarget Target_10230:=[[253.025190558,236.012109808,0],[0,0,1,0],[0,0,0,0],[9E+09,9E+09,9E+09,9E+09,9E+09,9E+09]];
    CONST robtarget Target_10240:=[[249.285935332,239.478831554,0],[0,0,1,0],[0,0,0,0],[9E+09,9E+09,9E+09,9E+09,9E+09,9E+09]];
    CONST robtarget Target_10250:=[[253.630423114,239.067306748,0],[0,0,1,0],[0,0,0,0],[9E+09,9E+09,9E+09,9E+09,9E+09,9E+09]];
    CONST robtarget Target_10260:=[[249.234575485,248.500819849,0],[0,0,1,0],[0,0,0,0],[9E+09,9E+09,9E+09,9E+09,9E+09,9E+09]];
    CONST robtarget Target_10270:=[[247.2072771,253.186666747,0],[0,0,1,0],[0,0,0,0],[9E+09,9E+09,9E+09,9E+09,9E+09,9E+09]];
    CONST robtarget Target_10280:=[[245.558776892,257.958629515,0],[0,0,1,0],[0,0,0,0],[9E+09,9E+09,9E+09,9E+09,9E+09,9E+09]];
    CONST robtarget Target_10290:=[[244.422181644,262.867346768,0],[0,0,1,0],[0,0,0,0],[9E+09,9E+09,9E+09,9E+09,9E+09,9E+09]];
    CONST robtarget Target_10300:=[[243.655887798,267.882591463,0],[0,0,1,0],[0,0,0,0],[9E+09,9E+09,9E+09,9E+09,9E+09,9E+09]];
    CONST robtarget Target_10310:=[[242.402489393,277.993398201,0],[0,0,1,0],[0,0,0,0],[9E+09,9E+09,9E+09,9E+09,9E+09,9E+09]];
    CONST robtarget Target_10320:=[[236.715389408,271.476863147,0],[0,0,1,0],[0,0,0,0],[9E+09,9E+09,9E+09,9E+09,9E+09,9E+09]];
    CONST robtarget Target_10330:=[[236.037033089,280.239056102,0],[0,0,1,0],[0,0,0,0],[9E+09,9E+09,9E+09,9E+09,9E+09,9E+09]];
    CONST robtarget Target_10340:=[[234.983545314,280.65358638,0],[0,0,1,0],[0,0,0,0],[9E+09,9E+09,9E+09,9E+09,9E+09,9E+09]];
    CONST robtarget Target_10350:=[[227.914134693,270.060106632,0],[0,0,1,0],[0,0,0,0],[9E+09,9E+09,9E+09,9E+09,9E+09,9E+09]];
    CONST robtarget Target_10360:=[[225.035155722,281.433267328,0],[0,0,1,0],[0,0,0,0],[9E+09,9E+09,9E+09,9E+09,9E+09,9E+09]];
    CONST robtarget Target_10370:=[[218.032445957,272.899415259,0],[0,0,1,0],[0,0,0,0],[9E+09,9E+09,9E+09,9E+09,9E+09,9E+09]];
    CONST robtarget Target_10380:=[[218.032445957,282.663881267,0],[0,0,1,0],[0,0,0,0],[9E+09,9E+09,9E+09,9E+09,9E+09,9E+09]];
    CONST robtarget Target_10390:=[[205.206687803,271.747889211,0],[0,0,1,0],[0,0,0,0],[9E+09,9E+09,9E+09,9E+09,9E+09,9E+09]];
    CONST robtarget Target_10400:=[[204.193722389,272.669538867,0],[0,0,1,0],[0,0,0,0],[9E+09,9E+09,9E+09,9E+09,9E+09,9E+09]];
    CONST robtarget Target_10410:=[[208.893953532,279.670465085,0],[0,0,1,0],[0,0,0,0],[9E+09,9E+09,9E+09,9E+09,9E+09,9E+09]];
    CONST robtarget Target_10420:=[[213.884830564,286.493752962,0],[0,0,1,0],[0,0,0,0],[9E+09,9E+09,9E+09,9E+09,9E+09,9E+09]];
    CONST robtarget Target_10430:=[[224.292532886,300.056031139,0],[0,0,1,0],[0,0,0,0],[9E+09,9E+09,9E+09,9E+09,9E+09,9E+09]];
    CONST robtarget Target_10440:=[[224.947450866,298.848905772,0],[0,0,1,0],[0,0,0,0],[9E+09,9E+09,9E+09,9E+09,9E+09,9E+09]];
    CONST robtarget Target_10450:=[[225.590271397,297.895057274,0],[0,0,1,0],[0,0,0,0],[9E+09,9E+09,9E+09,9E+09,9E+09,9E+09]];
    CONST robtarget Target_10460:=[[226.940295146,296.717509132,0],[0,0,1,0],[0,0,0,0],[9E+09,9E+09,9E+09,9E+09,9E+09,9E+09]];
    CONST robtarget Target_10470:=[[228.543954205,296.464023206,0],[0,0,1,0],[0,0,0,0],[9E+09,9E+09,9E+09,9E+09,9E+09,9E+09]];
    CONST robtarget Target_10480:=[[230.602598642,297.075235989,0],[0,0,1,0],[0,0,0,0],[9E+09,9E+09,9E+09,9E+09,9E+09,9E+09]];
    CONST robtarget Target_10490:=[[233.994404899,299.03285199,0],[0,0,1,0],[0,0,0,0],[9E+09,9E+09,9E+09,9E+09,9E+09,9E+09]];
    CONST robtarget Target_10500:=[[237.217200058,301.348664515,0],[0,0,1,0],[0,0,0,0],[9E+09,9E+09,9E+09,9E+09,9E+09,9E+09]];
    CONST robtarget Target_10510:=[[239.110951366,302.832139539,0],[0,0,1,0],[0,0,0,0],[9E+09,9E+09,9E+09,9E+09,9E+09,9E+09]];
    CONST robtarget Target_10520:=[[241.087029419,304.49834185,0],[0,0,1,0],[0,0,0,0],[9E+09,9E+09,9E+09,9E+09,9E+09,9E+09]];
    CONST robtarget Target_10530:=[[242.15079759,296.590208226,0],[0,0,1,0],[0,0,0,0],[9E+09,9E+09,9E+09,9E+09,9E+09,9E+09]];
    CONST robtarget Target_10540:=[[246.062050112,299.194172684,0],[0,0,1,0],[0,0,0,0],[9E+09,9E+09,9E+09,9E+09,9E+09,9E+09]];
    CONST robtarget Target_10550:=[[247.678787725,300.353785167,0],[0,0,1,0],[0,0,0,0],[9E+09,9E+09,9E+09,9E+09,9E+09,9E+09]];
    CONST robtarget Target_10560:=[[249.051414972,301.608656474,0],[0,0,1,0],[0,0,0,0],[9E+09,9E+09,9E+09,9E+09,9E+09,9E+09]];
    CONST robtarget Target_10570:=[[252.473494102,305.895493098,0],[0,0,1,0],[0,0,0,0],[9E+09,9E+09,9E+09,9E+09,9E+09,9E+09]];
    CONST robtarget Target_10580:=[[255.7169315,310.351894365,0],[0,0,1,0],[0,0,0,0],[9E+09,9E+09,9E+09,9E+09,9E+09,9E+09]];
    CONST robtarget Target_10590:=[[278.774941761,340.129287899,0],[0,0,1,0],[0,0,0,0],[9E+09,9E+09,9E+09,9E+09,9E+09,9E+09]];
    CONST robtarget Target_10600:=[[280.05315717,342.389221068,0],[0,0,1,0],[0,0,0,0],[9E+09,9E+09,9E+09,9E+09,9E+09,9E+09]];
    CONST robtarget Target_10610:=[[280.656646069,344.9487386,0],[0,0,1,0],[0,0,0,0],[9E+09,9E+09,9E+09,9E+09,9E+09,9E+09]];
    CONST robtarget Target_10620:=[[280.668475249,346.225027591,0],[0,0,1,0],[0,0,0,0],[9E+09,9E+09,9E+09,9E+09,9E+09,9E+09]];
    CONST robtarget Target_10630:=[[280.46735141,347.43723598,0],[0,0,1,0],[0,0,0,0],[9E+09,9E+09,9E+09,9E+09,9E+09,9E+09]];
    CONST robtarget Target_10640:=[[280.03851742,348.539038201,0],[0,0,1,0],[0,0,0,0],[9E+09,9E+09,9E+09,9E+09,9E+09,9E+09]];
    CONST robtarget Target_10650:=[[279.367216149,349.48410869,0],[0,0,1,0],[0,0,0,0],[9E+09,9E+09,9E+09,9E+09,9E+09,9E+09]];
    CONST robtarget Target_10660:=[[277.995759913,350.424910512,0],[0,0,1,0],[0,0,0,0],[9E+09,9E+09,9E+09,9E+09,9E+09,9E+09]];
    CONST robtarget Target_10670:=[[276.433314624,350.443600123,0],[0,0,1,0],[0,0,0,0],[9E+09,9E+09,9E+09,9E+09,9E+09,9E+09]];
    CONST robtarget Target_10680:=[[274.590134083,349.516586598,0],[0,0,1,0],[0,0,0,0],[9E+09,9E+09,9E+09,9E+09,9E+09,9E+09]];
    CONST robtarget Target_10690:=[[273.535222406,348.691068996,0],[0,0,1,0],[0,0,0,0],[9E+09,9E+09,9E+09,9E+09,9E+09,9E+09]];
    CONST robtarget Target_10700:=[[270.158022595,345.512538053,0],[0,0,1,0],[0,0,0,0],[9E+09,9E+09,9E+09,9E+09,9E+09,9E+09]];
    CONST robtarget Target_10710:=[[266.568479144,343.633449292,0],[0,0,1,0],[0,0,0,0],[9E+09,9E+09,9E+09,9E+09,9E+09,9E+09]];
    CONST robtarget Target_10720:=[[265.44549165,345.959997274,0],[0,0,1,0],[0,0,0,0],[9E+09,9E+09,9E+09,9E+09,9E+09,9E+09]];
    CONST robtarget Target_10730:=[[264.693155048,347.954007957,0],[0,0,1,0],[0,0,0,0],[9E+09,9E+09,9E+09,9E+09,9E+09,9E+09]];
    CONST robtarget Target_10740:=[[264.317913111,349.699450189,0],[0,0,1,0],[0,0,0,0],[9E+09,9E+09,9E+09,9E+09,9E+09,9E+09]];
    CONST robtarget Target_10750:=[[264.326209612,351.280292817,0],[0,0,1,0],[0,0,0,0],[9E+09,9E+09,9E+09,9E+09,9E+09,9E+09]];
    CONST robtarget Target_10760:=[[264.724488322,352.780504689,0],[0,0,1,0],[0,0,0,0],[9E+09,9E+09,9E+09,9E+09,9E+09,9E+09]];
    CONST robtarget Target_10770:=[[265.519193013,354.284054652,0],[0,0,1,0],[0,0,0,0],[9E+09,9E+09,9E+09,9E+09,9E+09,9E+09]];
    CONST robtarget Target_10780:=[[266.716767458,355.874911553,0],[0,0,1,0],[0,0,0,0],[9E+09,9E+09,9E+09,9E+09,9E+09,9E+09]];
    CONST robtarget Target_10790:=[[268.323655429,357.63704424,0],[0,0,1,0],[0,0,0,0],[9E+09,9E+09,9E+09,9E+09,9E+09,9E+09]];
    CONST robtarget Target_10800:=[[270.242856893,359.971268803,0],[0,0,1,0],[0,0,0,0],[9E+09,9E+09,9E+09,9E+09,9E+09,9E+09]];
    CONST robtarget Target_10810:=[[271.750266778,362.581653639,0],[0,0,1,0],[0,0,0,0],[9E+09,9E+09,9E+09,9E+09,9E+09,9E+09]];
    CONST robtarget Target_10820:=[[272.017414102,363.681313393,0],[0,0,1,0],[0,0,0,0],[9E+09,9E+09,9E+09,9E+09,9E+09,9E+09]];
    CONST robtarget Target_10830:=[[271.003781673,365.185546675,0],[0,0,1,0],[0,0,0,0],[9E+09,9E+09,9E+09,9E+09,9E+09,9E+09]];
    CONST robtarget Target_10840:=[[269.753697811,365.327724787,0],[0,0,1,0],[0,0,0,0],[9E+09,9E+09,9E+09,9E+09,9E+09,9E+09]];
    CONST robtarget Target_10850:=[[267.664723326,365.005310534,0],[0,0,1,0],[0,0,0,0],[9E+09,9E+09,9E+09,9E+09,9E+09,9E+09]];
    CONST robtarget Target_10860:=[[265.643805291,364.394593951,0],[0,0,1,0],[0,0,0,0],[9E+09,9E+09,9E+09,9E+09,9E+09,9E+09]];
    CONST robtarget Target_10870:=[[263.292362616,363.285076605,0],[0,0,1,0],[0,0,0,0],[9E+09,9E+09,9E+09,9E+09,9E+09,9E+09]];
    CONST robtarget Target_10880:=[[260.616523205,361.859641919,0],[0,0,1,0],[0,0,0,0],[9E+09,9E+09,9E+09,9E+09,9E+09,9E+09]];
    CONST robtarget Target_10890:=[[259.495248485,367.931642897,0],[0,0,1,0],[0,0,0,0],[9E+09,9E+09,9E+09,9E+09,9E+09,9E+09]];
    CONST robtarget Target_10900:=[[257.252208402,366.072413262,0],[0,0,1,0],[0,0,0,0],[9E+09,9E+09,9E+09,9E+09,9E+09,9E+09]];
    CONST robtarget Target_10910:=[[255.257497053,364.232360551,0],[0,0,1,0],[0,0,0,0],[9E+09,9E+09,9E+09,9E+09,9E+09,9E+09]];
    CONST robtarget Target_10920:=[[250.569617835,358.563908997,0],[0,0,1,0],[0,0,0,0],[9E+09,9E+09,9E+09,9E+09,9E+09,9E+09]];
    CONST robtarget Target_10930:=[[248.320898575,356.277123086,0],[0,0,1,0],[0,0,0,0],[9E+09,9E+09,9E+09,9E+09,9E+09,9E+09]];
    CONST robtarget Target_10940:=[[245.768469864,354.674541386,0],[0,0,1,0],[0,0,0,0],[9E+09,9E+09,9E+09,9E+09,9E+09,9E+09]];
    CONST robtarget Target_10950:=[[242.884192666,353.756031314,0],[0,0,1,0],[0,0,0,0],[9E+09,9E+09,9E+09,9E+09,9E+09,9E+09]];
    CONST robtarget Target_10960:=[[239.639927947,353.521460284,0],[0,0,1,0],[0,0,0,0],[9E+09,9E+09,9E+09,9E+09,9E+09,9E+09]];
    CONST robtarget Target_10970:=[[234.41447233,353.355702471,0],[0,0,1,0],[0,0,0,0],[9E+09,9E+09,9E+09,9E+09,9E+09,9E+09]];
    CONST robtarget Target_10980:=[[229.287005248,352.59141421,0],[0,0,1,0],[0,0,0,0],[9E+09,9E+09,9E+09,9E+09,9E+09,9E+09]];
    CONST robtarget Target_10990:=[[224.255176041,351.32286999,0],[0,0,1,0],[0,0,0,0],[9E+09,9E+09,9E+09,9E+09,9E+09,9E+09]];
    CONST robtarget Target_11000:=[[219.316634053,349.644344295,0],[0,0,1,0],[0,0,0,0],[9E+09,9E+09,9E+09,9E+09,9E+09,9E+09]];
    CONST robtarget Target_11010:=[[215.362585879,348.022941985,0],[0,0,1,0],[0,0,0,0],[9E+09,9E+09,9E+09,9E+09,9E+09,9E+09]];
    CONST robtarget Target_11020:=[[211.602587573,346.182593,0],[0,0,1,0],[0,0,0,0],[9E+09,9E+09,9E+09,9E+09,9E+09,9E+09]];
    CONST robtarget Target_11030:=[[208.081974825,344.075720932,0],[0,0,1,0],[0,0,0,0],[9E+09,9E+09,9E+09,9E+09,9E+09,9E+09]];
    CONST robtarget Target_11040:=[[204.846083322,341.654749375,0],[0,0,1,0],[0,0,0,0],[9E+09,9E+09,9E+09,9E+09,9E+09,9E+09]];
    CONST robtarget Target_11050:=[[201.940248752,338.87210192,0],[0,0,1,0],[0,0,0,0],[9E+09,9E+09,9E+09,9E+09,9E+09,9E+09]];
    CONST robtarget Target_11060:=[[199.409806803,335.680202161,0],[0,0,1,0],[0,0,0,0],[9E+09,9E+09,9E+09,9E+09,9E+09,9E+09]];
    CONST robtarget Target_11070:=[[197.300093164,332.03147369,0],[0,0,1,0],[0,0,0,0],[9E+09,9E+09,9E+09,9E+09,9E+09,9E+09]];
    CONST robtarget Target_11080:=[[195.20679628,326.729446882,0],[0,0,1,0],[0,0,0,0],[9E+09,9E+09,9E+09,9E+09,9E+09,9E+09]];
    CONST robtarget Target_11090:=[[194.554418796,325.704996075,0],[0,0,1,0],[0,0,0,0],[9E+09,9E+09,9E+09,9E+09,9E+09,9E+09]];
    CONST robtarget Target_11100:=[[192.267320975,323.719423761,0],[0,0,1,0],[0,0,0,0],[9E+09,9E+09,9E+09,9E+09,9E+09,9E+09]];
    CONST robtarget Target_11110:=[[190.439264361,327.056100372,0],[0,0,1,0],[0,0,0,0],[9E+09,9E+09,9E+09,9E+09,9E+09,9E+09]];
    CONST robtarget Target_11120:=[[174.175097682,315.242862896,0],[0,0,1,0],[0,0,0,0],[9E+09,9E+09,9E+09,9E+09,9E+09,9E+09]];
    CONST robtarget Target_11130:=[[176.498324353,314.725148515,0],[0,0,1,0],[0,0,0,0],[9E+09,9E+09,9E+09,9E+09,9E+09,9E+09]];
    CONST robtarget Target_11140:=[[178.687358153,314.382672662,0],[0,0,1,0],[0,0,0,0],[9E+09,9E+09,9E+09,9E+09,9E+09,9E+09]];
    CONST robtarget Target_11150:=[[182.842445091,314.125834223,0],[0,0,1,0],[0,0,0,0],[9E+09,9E+09,9E+09,9E+09,9E+09,9E+09]];
    CONST robtarget Target_11160:=[[186.789618222,314.093444437,0],[0,0,1,0],[0,0,0,0],[9E+09,9E+09,9E+09,9E+09,9E+09,9E+09]];
    CONST robtarget Target_11170:=[[188.04185962,314.046141324,0],[0,0,1,0],[0,0,0,0],[9E+09,9E+09,9E+09,9E+09,9E+09,9E+09]];
    CONST robtarget Target_11180:=[[190.037260683,313.574226077,0],[0,0,1,0],[0,0,0,0],[9E+09,9E+09,9E+09,9E+09,9E+09,9E+09]];
    CONST robtarget Target_11190:=[[190.836473389,312.813300136,0],[0,0,1,0],[0,0,0,0],[9E+09,9E+09,9E+09,9E+09,9E+09,9E+09]];
    CONST robtarget Target_11200:=[[180.856521671,310.771855088,0],[0,0,1,0],[0,0,0,0],[9E+09,9E+09,9E+09,9E+09,9E+09,9E+09]];
    CONST robtarget Target_11210:=[[178.374933216,310.178378557,0],[0,0,1,0],[0,0,0,0],[9E+09,9E+09,9E+09,9E+09,9E+09,9E+09]];
    CONST robtarget Target_11220:=[[175.941894623,309.308468352,0],[0,0,1,0],[0,0,0,0],[9E+09,9E+09,9E+09,9E+09,9E+09,9E+09]];
    CONST robtarget Target_11230:=[[173.598895413,307.913844129,0],[0,0,1,0],[0,0,0,0],[9E+09,9E+09,9E+09,9E+09,9E+09,9E+09]];
    CONST robtarget Target_11240:=[[172.474126051,306.942176653,0],[0,0,1,0],[0,0,0,0],[9E+09,9E+09,9E+09,9E+09,9E+09,9E+09]];
    CONST robtarget Target_11250:=[[171.387425105,305.746225543,0],[0,0,1,0],[0,0,0,0],[9E+09,9E+09,9E+09,9E+09,9E+09,9E+09]];
    CONST robtarget Target_11260:=[[176.181184152,306.061118465,0],[0,0,1,0],[0,0,0,0],[9E+09,9E+09,9E+09,9E+09,9E+09,9E+09]];
    CONST robtarget Target_11270:=[[180.333260759,306.532315353,0],[0,0,1,0],[0,0,0,0],[9E+09,9E+09,9E+09,9E+09,9E+09,9E+09]];
    CONST robtarget Target_11280:=[[184.504288115,307.493093058,0],[0,0,1,0],[0,0,0,0],[9E+09,9E+09,9E+09,9E+09,9E+09,9E+09]];
    CONST robtarget Target_11290:=[[188.536866816,308.892499486,0],[0,0,1,0],[0,0,0,0],[9E+09,9E+09,9E+09,9E+09,9E+09,9E+09]];
    CONST robtarget Target_11300:=[[191.739912326,310.681704419,0],[0,0,1,0],[0,0,0,0],[9E+09,9E+09,9E+09,9E+09,9E+09,9E+09]];
    CONST robtarget Target_11310:=[[194.828469056,312.741566755,0],[0,0,1,0],[0,0,0,0],[9E+09,9E+09,9E+09,9E+09,9E+09,9E+09]];
    CONST robtarget Target_11320:=[[192.133507298,308.543551206,0],[0,0,1,0],[0,0,0,0],[9E+09,9E+09,9E+09,9E+09,9E+09,9E+09]];
    CONST robtarget Target_11330:=[[195.23457278,307.816058715,0],[0,0,1,0],[0,0,0,0],[9E+09,9E+09,9E+09,9E+09,9E+09,9E+09]];
    CONST robtarget Target_11340:=[[195.777842076,306.947880224,0],[0,0,1,0],[0,0,0,0],[9E+09,9E+09,9E+09,9E+09,9E+09,9E+09]];
    CONST robtarget Target_11350:=[[193.025167786,305.03007613,0],[0,0,1,0],[0,0,0,0],[9E+09,9E+09,9E+09,9E+09,9E+09,9E+09]];
    CONST robtarget Target_11360:=[[188.248440986,300.010267872,0],[0,0,1,0],[0,0,0,0],[9E+09,9E+09,9E+09,9E+09,9E+09,9E+09]];
    CONST robtarget Target_11370:=[[183.919399947,294.672489256,0],[0,0,1,0],[0,0,0,0],[9E+09,9E+09,9E+09,9E+09,9E+09,9E+09]];
    CONST robtarget Target_11380:=[[181.997132854,291.842412552,0],[0,0,1,0],[0,0,0,0],[9E+09,9E+09,9E+09,9E+09,9E+09,9E+09]];
    CONST robtarget Target_11390:=[[180.27603272,288.882505045,0],[0,0,1,0],[0,0,0,0],[9E+09,9E+09,9E+09,9E+09,9E+09,9E+09]];
    CONST robtarget Target_11400:=[[178.785848052,285.775987329,0],[0,0,1,0],[0,0,0,0],[9E+09,9E+09,9E+09,9E+09,9E+09,9E+09]];
    CONST robtarget Target_11410:=[[177.556327357,282.50608,0],[0,0,1,0],[0,0,0,0],[9E+09,9E+09,9E+09,9E+09,9E+09,9E+09]];
    CONST robtarget Target_11420:=[[176.22245259,279.251954792,0],[0,0,1,0],[0,0,0,0],[9E+09,9E+09,9E+09,9E+09,9E+09,9E+09]];
    CONST robtarget Target_11430:=[[174.497548762,276.330610095,0],[0,0,1,0],[0,0,0,0],[9E+09,9E+09,9E+09,9E+09,9E+09,9E+09]];
    CONST robtarget Target_11440:=[[172.439747083,273.657279757,0],[0,0,1,0],[0,0,0,0],[9E+09,9E+09,9E+09,9E+09,9E+09,9E+09]];
    CONST robtarget Target_11450:=[[166.148402444,266.878970162,0],[0,0,1,0],[0,0,0,0],[9E+09,9E+09,9E+09,9E+09,9E+09,9E+09]];
    CONST robtarget Target_11460:=[[164.504535069,264.422237091,0],[0,0,1,0],[0,0,0,0],[9E+09,9E+09,9E+09,9E+09,9E+09,9E+09]];
    CONST robtarget Target_11470:=[[162.795148928,261.595904712,0],[0,0,1,0],[0,0,0,0],[9E+09,9E+09,9E+09,9E+09,9E+09,9E+09]];
    CONST robtarget Target_11480:=[[164.964546517,261.997261477,0],[0,0,1,0],[0,0,0,0],[9E+09,9E+09,9E+09,9E+09,9E+09,9E+09]];
    CONST robtarget Target_11490:=[[164.421010947,259.676274554,0],[0,0,1,0],[0,0,0,0],[9E+09,9E+09,9E+09,9E+09,9E+09,9E+09]];
    CONST robtarget Target_11500:=[[163.632675097,257.508603403,0],[0,0,1,0],[0,0,0,0],[9E+09,9E+09,9E+09,9E+09,9E+09,9E+09]];
    CONST robtarget Target_11510:=[[162.633037044,255.476885703,0],[0,0,1,0],[0,0,0,0],[9E+09,9E+09,9E+09,9E+09,9E+09,9E+09]];
    CONST robtarget Target_11520:=[[161.455594862,253.563759132,0],[0,0,1,0],[0,0,0,0],[9E+09,9E+09,9E+09,9E+09,9E+09,9E+09]];
    CONST robtarget Target_11530:=[[158.701290414,250.02383009,0],[0,0,1,0],[0,0,0,0],[9E+09,9E+09,9E+09,9E+09,9E+09,9E+09]];
    CONST robtarget Target_11540:=[[152.516444237,243.34696935,0],[0,0,1,0],[0,0,0,0],[9E+09,9E+09,9E+09,9E+09,9E+09,9E+09]];
    CONST robtarget Target_11550:=[[149.652862782,239.790230466,0],[0,0,1,0],[0,0,0,0],[9E+09,9E+09,9E+09,9E+09,9E+09,9E+09]];
    CONST robtarget Target_11560:=[[147.018073238,236.09599875,0],[0,0,1,0],[0,0,0,0],[9E+09,9E+09,9E+09,9E+09,9E+09,9E+09]];
    CONST robtarget Target_11570:=[[144.583146852,232.280571901,0],[0,0,1,0],[0,0,0,0],[9E+09,9E+09,9E+09,9E+09,9E+09,9E+09]];
    CONST robtarget Target_11580:=[[140.197168532,224.351323615,0],[0,0,1,0],[0,0,0,0],[9E+09,9E+09,9E+09,9E+09,9E+09,9E+09]];
    CONST robtarget Target_11590:=[[136.263497785,216.132867219,0],[0,0,1,0],[0,0,0,0],[9E+09,9E+09,9E+09,9E+09,9E+09,9E+09]];
    CONST robtarget Target_11600:=[[134.595264811,211.537249404,0],[0,0,1,0],[0,0,0,0],[9E+09,9E+09,9E+09,9E+09,9E+09,9E+09]];
    CONST robtarget Target_11610:=[[133.353237573,207.125124482,0],[0,0,1,0],[0,0,0,0],[9E+09,9E+09,9E+09,9E+09,9E+09,9E+09]];
    CONST robtarget Target_11620:=[[132.476426546,202.701277287,0],[0,0,1,0],[0,0,0,0],[9E+09,9E+09,9E+09,9E+09,9E+09,9E+09]];
    CONST robtarget Target_11630:=[[134.856811367,205.64410655,0],[0,0,1,0],[0,0,0,0],[9E+09,9E+09,9E+09,9E+09,9E+09,9E+09]];
    CONST robtarget Target_11640:=[[137.425256244,208.245898144,0],[0,0,1,0],[0,0,0,0],[9E+09,9E+09,9E+09,9E+09,9E+09,9E+09]];
    CONST robtarget Target_11650:=[[140.175223138,210.523832472,0],[0,0,1,0],[0,0,0,0],[9E+09,9E+09,9E+09,9E+09,9E+09,9E+09]];
    CONST robtarget Target_11660:=[[143.100174008,212.495089939,0],[0,0,1,0],[0,0,0,0],[9E+09,9E+09,9E+09,9E+09,9E+09,9E+09]];
    CONST robtarget Target_11670:=[[146.193570813,214.176850952,0],[0,0,1,0],[0,0,0,0],[9E+09,9E+09,9E+09,9E+09,9E+09,9E+09]];
    CONST robtarget Target_11680:=[[149.448875514,215.586295914,0],[0,0,1,0],[0,0,0,0],[9E+09,9E+09,9E+09,9E+09,9E+09,9E+09]];
    CONST robtarget Target_11690:=[[152.85955007,216.74060523,0],[0,0,1,0],[0,0,0,0],[9E+09,9E+09,9E+09,9E+09,9E+09,9E+09]];
    CONST robtarget Target_11700:=[[156.41905644,217.656959306,0],[0,0,1,0],[0,0,0,0],[9E+09,9E+09,9E+09,9E+09,9E+09,9E+09]];
    CONST robtarget Target_11710:=[[153.622357609,215.389456275,0],[0,0,1,0],[0,0,0,0],[9E+09,9E+09,9E+09,9E+09,9E+09,9E+09]];
    CONST robtarget Target_11720:=[[150.985204275,212.97868863,0],[0,0,1,0],[0,0,0,0],[9E+09,9E+09,9E+09,9E+09,9E+09,9E+09]];
    CONST robtarget Target_11730:=[[146.089729734,207.817253348,0],[0,0,1,0],[0,0,0,0],[9E+09,9E+09,9E+09,9E+09,9E+09,9E+09]];
    CONST robtarget Target_11740:=[[137.115478566,196.764039729,0],[0,0,1,0],[0,0,0,0],[9E+09,9E+09,9E+09,9E+09,9E+09,9E+09]];
    CONST robtarget Target_11750:=[[131.03310766,189.066214166,0],[0,0,1,0],[0,0,0,0],[9E+09,9E+09,9E+09,9E+09,9E+09,9E+09]];
    CONST robtarget Target_11760:=[[124.720390994,181.83127057,0],[0,0,1,0],[0,0,0,0],[9E+09,9E+09,9E+09,9E+09,9E+09,9E+09]];
    CONST robtarget Target_11770:=[[121.343550391,178.496989466,0],[0,0,1,0],[0,0,0,0],[9E+09,9E+09,9E+09,9E+09,9E+09,9E+09]];
    CONST robtarget Target_11780:=[[117.773863853,175.43373072,0],[0,0,1,0],[0,0,0,0],[9E+09,9E+09,9E+09,9E+09,9E+09,9E+09]];
    CONST robtarget Target_11790:=[[113.976938064,172.703165757,0],[0,0,1,0],[0,0,0,0],[9E+09,9E+09,9E+09,9E+09,9E+09,9E+09]];
    CONST robtarget Target_11800:=[[109.918379707,170.366965999,0],[0,0,1,0],[0,0,0,0],[9E+09,9E+09,9E+09,9E+09,9E+09,9E+09]];
    CONST robtarget Target_11810:=[[105.563795467,168.486802869,0],[0,0,1,0],[0,0,0,0],[9E+09,9E+09,9E+09,9E+09,9E+09,9E+09]];
    CONST robtarget Target_11820:=[[100.878792027,167.12434779,0],[0,0,1,0],[0,0,0,0],[9E+09,9E+09,9E+09,9E+09,9E+09,9E+09]];
    CONST robtarget Target_11830:=[[97.924657366,166.350586532,0],[0,0,1,0],[0,0,0,0],[9E+09,9E+09,9E+09,9E+09,9E+09,9E+09]];
    CONST robtarget Target_11840:=[[95.116630976,165.386476662,0],[0,0,1,0],[0,0,0,0],[9E+09,9E+09,9E+09,9E+09,9E+09,9E+09]];
    CONST robtarget Target_11850:=[[92.439571996,164.241298142,0],[0,0,1,0],[0,0,0,0],[9E+09,9E+09,9E+09,9E+09,9E+09,9E+09]];
    CONST robtarget Target_11860:=[[89.878339567,162.924330934,0],[0,0,1,0],[0,0,0,0],[9E+09,9E+09,9E+09,9E+09,9E+09,9E+09]];
    CONST robtarget Target_11870:=[[85.042790916,159.812150301,0],[0,0,1,0],[0,0,0,0],[9E+09,9E+09,9E+09,9E+09,9E+09,9E+09]];
    CONST robtarget Target_11880:=[[75.030520364,151.658569008,0],[0,0,1,0],[0,0,0,0],[9E+09,9E+09,9E+09,9E+09,9E+09,9E+09]];
    CONST robtarget Target_11890:=[[70.782575713,148.008694142,0],[0,0,1,0],[0,0,0,0],[9E+09,9E+09,9E+09,9E+09,9E+09,9E+09]];
    CONST robtarget Target_11900:=[[66.694726875,144.225670247,0],[0,0,1,0],[0,0,0,0],[9E+09,9E+09,9E+09,9E+09,9E+09,9E+09]];
    CONST robtarget Target_11910:=[[62.802088788,140.284357775,0],[0,0,1,0],[0,0,0,0],[9E+09,9E+09,9E+09,9E+09,9E+09,9E+09]];
    CONST robtarget Target_11920:=[[59.139776387,136.159617175,0],[0,0,1,0],[0,0,0,0],[9E+09,9E+09,9E+09,9E+09,9E+09,9E+09]];
    CONST robtarget Target_11930:=[[55.74290461,131.826308896,0],[0,0,1,0],[0,0,0,0],[9E+09,9E+09,9E+09,9E+09,9E+09,9E+09]];
    CONST robtarget Target_11940:=[[52.646588392,127.259293388,0],[0,0,1,0],[0,0,0,0],[9E+09,9E+09,9E+09,9E+09,9E+09,9E+09]];
    CONST robtarget Target_11950:=[[49.885942671,122.433431101,0],[0,0,1,0],[0,0,0,0],[9E+09,9E+09,9E+09,9E+09,9E+09,9E+09]];
    CONST robtarget Target_11960:=[[47.496082383,117.323582483,0],[0,0,1,0],[0,0,0,0],[9E+09,9E+09,9E+09,9E+09,9E+09,9E+09]];
    CONST robtarget Target_11970:=[[45.992283919,113.551179016,0],[0,0,1,0],[0,0,0,0],[9E+09,9E+09,9E+09,9E+09,9E+09,9E+09]];
    CONST robtarget Target_11980:=[[44.690574674,109.656732056,0],[0,0,1,0],[0,0,0,0],[9E+09,9E+09,9E+09,9E+09,9E+09,9E+09]];
    CONST robtarget Target_11990:=[[43.79654362,105.717992757,0],[0,0,1,0],[0,0,0,0],[9E+09,9E+09,9E+09,9E+09,9E+09,9E+09]];
    CONST robtarget Target_12000:=[[43.515779729,101.812712276,0],[0,0,1,0],[0,0,0,0],[9E+09,9E+09,9E+09,9E+09,9E+09,9E+09]];
    CONST robtarget Target_12010:=[[43.409764153,96.908920753,0],[0,0,1,0],[0,0,0,0],[9E+09,9E+09,9E+09,9E+09,9E+09,9E+09]];
    CONST robtarget Target_12020:=[[42.791617629,92.2158317,0],[0,0,1,0],[0,0,0,0],[9E+09,9E+09,9E+09,9E+09,9E+09,9E+09]];
    CONST robtarget Target_12030:=[[41.579665234,87.68366174,0],[0,0,1,0],[0,0,0,0],[9E+09,9E+09,9E+09,9E+09,9E+09,9E+09]];
    CONST robtarget Target_12040:=[[39.692232045,83.262627493,0],[0,0,1,0],[0,0,0,0],[9E+09,9E+09,9E+09,9E+09,9E+09,9E+09]];
    CONST robtarget Target_12050:=[[38.608715894,80.081921713,0],[0,0,1,0],[0,0,0,0],[9E+09,9E+09,9E+09,9E+09,9E+09,9E+09]];
    CONST robtarget Target_12060:=[[38.181534771,77.754883658,0],[0,0,1,0],[0,0,0,0],[9E+09,9E+09,9E+09,9E+09,9E+09,9E+09]];
    CONST robtarget Target_12070:=[[38.104787203,75.364902654,0],[0,0,1,0],[0,0,0,0],[9E+09,9E+09,9E+09,9E+09,9E+09,9E+09]];
    CONST robtarget Target_12080:=[[38.357053412,72.983005257,0],[0,0,1,0],[0,0,0,0],[9E+09,9E+09,9E+09,9E+09,9E+09,9E+09]];
    CONST robtarget Target_12090:=[[38.916913618,70.680218022,0],[0,0,1,0],[0,0,0,0],[9E+09,9E+09,9E+09,9E+09,9E+09,9E+09]];
    CONST robtarget Target_12100:=[[39.762948042,68.527567505,0],[0,0,1,0],[0,0,0,0],[9E+09,9E+09,9E+09,9E+09,9E+09,9E+09]];
    CONST robtarget Target_12110:=[[40.873736903,66.596080262,0],[0,0,1,0],[0,0,0,0],[9E+09,9E+09,9E+09,9E+09,9E+09,9E+09]];
    CONST robtarget Target_12120:=[[42.227860423,64.956782847,0],[0,0,1,0],[0,0,0,0],[9E+09,9E+09,9E+09,9E+09,9E+09,9E+09]];
    CONST robtarget Target_12130:=[[43.803898823,63.680701815,0],[0,0,1,0],[0,0,0,0],[9E+09,9E+09,9E+09,9E+09,9E+09,9E+09]];
    CONST robtarget Target_12140:=[[44.206514304,73.390701856,0],[0,0,1,0],[0,0,0,0],[9E+09,9E+09,9E+09,9E+09,9E+09,9E+09]];
    CONST robtarget Target_12150:=[[44.869361192,78.158429987,0],[0,0,1,0],[0,0,0,0],[9E+09,9E+09,9E+09,9E+09,9E+09,9E+09]];
    CONST robtarget Target_12160:=[[45.485262175,80.497277274,0],[0,0,1,0],[0,0,0,0],[9E+09,9E+09,9E+09,9E+09,9E+09,9E+09]];
    CONST robtarget Target_12170:=[[46.355231139,82.797275732,0],[0,0,1,0],[0,0,0,0],[9E+09,9E+09,9E+09,9E+09,9E+09,9E+09]];
    CONST robtarget Target_12180:=[[47.10711075,74.695890797,0],[0,0,1,0],[0,0,0,0],[9E+09,9E+09,9E+09,9E+09,9E+09,9E+09]];
    CONST robtarget Target_12190:=[[47.546592551,66.628029502,0],[0,0,1,0],[0,0,0,0],[9E+09,9E+09,9E+09,9E+09,9E+09,9E+09]];
    CONST robtarget Target_12200:=[[48.12956496,60.892316762,0],[0,0,1,0],[0,0,0,0],[9E+09,9E+09,9E+09,9E+09,9E+09,9E+09]];
    CONST robtarget Target_12210:=[[49.333946664,55.328511365,0],[0,0,1,0],[0,0,0,0],[9E+09,9E+09,9E+09,9E+09,9E+09,9E+09]];
    CONST robtarget Target_12220:=[[51.121442635,49.916723761,0],[0,0,1,0],[0,0,0,0],[9E+09,9E+09,9E+09,9E+09,9E+09,9E+09]];
    CONST robtarget Target_12230:=[[53.453757845,44.637064405,0],[0,0,1,0],[0,0,0,0],[9E+09,9E+09,9E+09,9E+09,9E+09,9E+09]];
    CONST robtarget Target_12240:=[[54.448927571,42.860544415,0],[0,0,1,0],[0,0,0,0],[9E+09,9E+09,9E+09,9E+09,9E+09,9E+09]];
    CONST robtarget Target_12250:=[[55.573976696,41.282581252,0],[0,0,1,0],[0,0,0,0],[9E+09,9E+09,9E+09,9E+09,9E+09,9E+09]];
    CONST robtarget Target_12260:=[[56.832229951,39.903404903,0],[0,0,1,0],[0,0,0,0],[9E+09,9E+09,9E+09,9E+09,9E+09,9E+09]];
    CONST robtarget Target_12270:=[[58.227012065,38.723245351,0],[0,0,1,0],[0,0,0,0],[9E+09,9E+09,9E+09,9E+09,9E+09,9E+09]];
    CONST robtarget Target_12280:=[[59.761647768,37.742332582,0],[0,0,1,0],[0,0,0,0],[9E+09,9E+09,9E+09,9E+09,9E+09,9E+09]];
    CONST robtarget Target_12290:=[[61.43946179,36.96089658,0],[0,0,1,0],[0,0,0,0],[9E+09,9E+09,9E+09,9E+09,9E+09,9E+09]];
    CONST robtarget Target_12300:=[[63.263778861,36.379167331,0],[0,0,1,0],[0,0,0,0],[9E+09,9E+09,9E+09,9E+09,9E+09,9E+09]];
    CONST robtarget Target_12310:=[[65.237923711,35.997374818,0],[0,0,1,0],[0,0,0,0],[9E+09,9E+09,9E+09,9E+09,9E+09,9E+09]];
    CONST robtarget Target_12320:=[[72.549930138,35.265388165,0],[0,0,1,0],[0,0,0,0],[9E+09,9E+09,9E+09,9E+09,9E+09,9E+09]];
    CONST robtarget Target_12330:=[[75.506188744,35.331819795,0],[0,0,1,0],[0,0,0,0],[9E+09,9E+09,9E+09,9E+09,9E+09,9E+09]];
    CONST robtarget Target_12340:=[[78.362735188,35.719243267,0],[0,0,1,0],[0,0,0,0],[9E+09,9E+09,9E+09,9E+09,9E+09,9E+09]];
    CONST robtarget Target_12350:=[[81.131571439,36.384084112,0],[0,0,1,0],[0,0,0,0],[9E+09,9E+09,9E+09,9E+09,9E+09,9E+09]];
    CONST robtarget Target_12360:=[[83.824699466,37.282767861,0],[0,0,1,0],[0,0,0,0],[9E+09,9E+09,9E+09,9E+09,9E+09,9E+09]];
    CONST robtarget Target_12370:=[[89.031838725,39.607366193,0],[0,0,1,0],[0,0,0,0],[9E+09,9E+09,9E+09,9E+09,9E+09,9E+09]];
    CONST robtarget Target_12380:=[[97.367547577,44.084981366,0],[0,0,1,0],[0,0,0,0],[9E+09,9E+09,9E+09,9E+09,9E+09,9E+09]];
    CONST robtarget Target_12390:=[[100.71323416,45.627688429,0],[0,0,1,0],[0,0,0,0],[9E+09,9E+09,9E+09,9E+09,9E+09,9E+09]];
    CONST robtarget Target_12400:=[[107.572238924,48.145231906,0],[0,0,1,0],[0,0,0,0],[9E+09,9E+09,9E+09,9E+09,9E+09,9E+09]];
    CONST robtarget Target_12410:=[[114.642599875,49.948322408,0],[0,0,1,0],[0,0,0,0],[9E+09,9E+09,9E+09,9E+09,9E+09,9E+09]];
    CONST robtarget Target_12420:=[[121.909733877,51.0882094,0],[0,0,1,0],[0,0,0,0],[9E+09,9E+09,9E+09,9E+09,9E+09,9E+09]];
    CONST robtarget Target_12430:=[[140.137886848,52.395898219,0],[0,0,1,0],[0,0,0,0],[9E+09,9E+09,9E+09,9E+09,9E+09,9E+09]];
    CONST robtarget Target_12440:=[[143.967305483,52.940417158,0],[0,0,1,0],[0,0,0,0],[9E+09,9E+09,9E+09,9E+09,9E+09,9E+09]];
    CONST robtarget Target_12450:=[[145.78535312,53.39850666,0],[0,0,1,0],[0,0,0,0],[9E+09,9E+09,9E+09,9E+09,9E+09,9E+09]];
    CONST robtarget Target_12460:=[[147.510968768,54.045463512,0],[0,0,1,0],[0,0,0,0],[9E+09,9E+09,9E+09,9E+09,9E+09,9E+09]];
    CONST robtarget Target_12470:=[[149.123159276,54.93002321,0],[0,0,1,0],[0,0,0,0],[9E+09,9E+09,9E+09,9E+09,9E+09,9E+09]];
    CONST robtarget Target_12480:=[[150.600931494,56.100921251,0],[0,0,1,0],[0,0,0,0],[9E+09,9E+09,9E+09,9E+09,9E+09,9E+09]];
    CONST robtarget Target_12490:=[[151.923292268,57.606893131,0],[0,0,1,0],[0,0,0,0],[9E+09,9E+09,9E+09,9E+09,9E+09,9E+09]];
    CONST robtarget Target_12500:=[[153.069248449,59.496674346,0],[0,0,1,0],[0,0,0,0],[9E+09,9E+09,9E+09,9E+09,9E+09,9E+09]];
    CONST robtarget Target_12510:=[[156.159469865,64.815456181,0],[0,0,1,0],[0,0,0,0],[9E+09,9E+09,9E+09,9E+09,9E+09,9E+09]];
    CONST robtarget Target_12520:=[[159.838678828,69.651065321,0],[0,0,1,0],[0,0,0,0],[9E+09,9E+09,9E+09,9E+09,9E+09,9E+09]];
    CONST robtarget Target_12530:=[[164.105124775,74.0646538,0],[0,0,1,0],[0,0,0,0],[9E+09,9E+09,9E+09,9E+09,9E+09,9E+09]];
    CONST robtarget Target_12540:=[[173.170575466,81.679242779,0],[0,0,1,0],[0,0,0,0],[9E+09,9E+09,9E+09,9E+09,9E+09,9E+09]];
    CONST robtarget Target_12550:=[[176.892821347,85.582430642,0],[0,0,1,0],[0,0,0,0],[9E+09,9E+09,9E+09,9E+09,9E+09,9E+09]];
    CONST robtarget Target_12560:=[[180.152283691,89.797944311,0],[0,0,1,0],[0,0,0,0],[9E+09,9E+09,9E+09,9E+09,9E+09,9E+09]];
    CONST robtarget Target_12570:=[[182.977451402,94.296790858,0],[0,0,1,0],[0,0,0,0],[9E+09,9E+09,9E+09,9E+09,9E+09,9E+09]];
    CONST robtarget Target_12580:=[[185.396813386,99.049977354,0],[0,0,1,0],[0,0,0,0],[9E+09,9E+09,9E+09,9E+09,9E+09,9E+09]];
    CONST robtarget Target_12590:=[[187.438858549,104.028510872,0],[0,0,1,0],[0,0,0,0],[9E+09,9E+09,9E+09,9E+09,9E+09,9E+09]];
    CONST robtarget Target_12600:=[[189.132075795,109.203398482,0],[0,0,1,0],[0,0,0,0],[9E+09,9E+09,9E+09,9E+09,9E+09,9E+09]];
    CONST robtarget Target_12610:=[[190.504954031,114.545647257,0],[0,0,1,0],[0,0,0,0],[9E+09,9E+09,9E+09,9E+09,9E+09,9E+09]];
    CONST robtarget Target_12620:=[[191.623648257,120.812709733,0],[0,0,1,0],[0,0,0,0],[9E+09,9E+09,9E+09,9E+09,9E+09,9E+09]];
    CONST robtarget Target_12630:=[[192.541202704,127.12516278,0],[0,0,1,0],[0,0,0,0],[9E+09,9E+09,9E+09,9E+09,9E+09,9E+09]];
    CONST robtarget Target_12640:=[[185.498139108,118.555881733,0],[0,0,1,0],[0,0,0,0],[9E+09,9E+09,9E+09,9E+09,9E+09,9E+09]];
    CONST robtarget Target_12650:=[[190.367357768,117.289745188,0],[0,0,1,0],[0,0,0,0],[9E+09,9E+09,9E+09,9E+09,9E+09,9E+09]];
    CONST robtarget Target_12660:=[[189.138434437,116.357802413,0],[0,0,1,0],[0,0,0,0],[9E+09,9E+09,9E+09,9E+09,9E+09,9E+09]];
    CONST robtarget Target_12670:=[[187.930525626,115.63633243,0],[0,0,1,0],[0,0,0,0],[9E+09,9E+09,9E+09,9E+09,9E+09,9E+09]];
    CONST robtarget Target_12680:=[[185.506762282,114.709496917,0],[0,0,1,0],[0,0,0,0],[9E+09,9E+09,9E+09,9E+09,9E+09,9E+09]];
    CONST robtarget Target_12690:=[[181.532650385,113.302508037,0],[0,0,1,0],[0,0,0,0],[9E+09,9E+09,9E+09,9E+09,9E+09,9E+09]];
    CONST robtarget Target_12700:=[[177.994002766,111.276666435,0],[0,0,1,0],[0,0,0,0],[9E+09,9E+09,9E+09,9E+09,9E+09,9E+09]];
    CONST robtarget Target_12710:=[[174.884173016,108.655138795,0],[0,0,1,0],[0,0,0,0],[9E+09,9E+09,9E+09,9E+09,9E+09,9E+09]];
    CONST robtarget Target_12720:=[[172.196514726,105.461091799,0],[0,0,1,0],[0,0,0,0],[9E+09,9E+09,9E+09,9E+09,9E+09,9E+09]];
    CONST robtarget Target_12730:=[[166.736193175,97.858309257,0],[0,0,1,0],[0,0,0,0],[9E+09,9E+09,9E+09,9E+09,9E+09,9E+09]];
    CONST robtarget Target_12740:=[[164.147743808,93.972660262,0],[0,0,1,0],[0,0,0,0],[9E+09,9E+09,9E+09,9E+09,9E+09,9E+09]];
    CONST robtarget Target_12750:=[[160.523540505,87.781678549,0],[0,0,1,0],[0,0,0,0],[9E+09,9E+09,9E+09,9E+09,9E+09,9E+09]];
    CONST robtarget Target_12760:=[[159.105081277,85.760696773,0],[0,0,1,0],[0,0,0,0],[9E+09,9E+09,9E+09,9E+09,9E+09,9E+09]];
    CONST robtarget Target_12770:=[[155.913895987,82.104777893,0],[0,0,1,0],[0,0,0,0],[9E+09,9E+09,9E+09,9E+09,9E+09,9E+09]];
    CONST robtarget Target_12780:=[[152.352957144,78.830518185,0],[0,0,1,0],[0,0,0,0],[9E+09,9E+09,9E+09,9E+09,9E+09,9E+09]];
    CONST robtarget Target_12790:=[[148.545387422,75.778237178,0],[0,0,1,0],[0,0,0,0],[9E+09,9E+09,9E+09,9E+09,9E+09,9E+09]];
    CONST robtarget Target_12800:=[[147.375739896,75.266491474,0],[0,0,1,0],[0,0,0,0],[9E+09,9E+09,9E+09,9E+09,9E+09,9E+09]];
    CONST robtarget Target_12810:=[[146.095516667,74.936386987,0],[0,0,1,0],[0,0,0,0],[9E+09,9E+09,9E+09,9E+09,9E+09,9E+09]];
    CONST robtarget Target_12820:=[[151.795558346,82.990883679,0],[0,0,1,0],[0,0,0,0],[9E+09,9E+09,9E+09,9E+09,9E+09,9E+09]];
    CONST robtarget Target_12830:=[[157.265016917,90.933282101,0],[0,0,1,0],[0,0,0,0],[9E+09,9E+09,9E+09,9E+09,9E+09,9E+09]];
    CONST robtarget Target_12840:=[[162.4556383,99.068746272,0],[0,0,1,0],[0,0,0,0],[9E+09,9E+09,9E+09,9E+09,9E+09,9E+09]];
    CONST robtarget Target_12850:=[[167.674442001,107.483652003,0],[0,0,1,0],[0,0,0,0],[9E+09,9E+09,9E+09,9E+09,9E+09,9E+09]];
    CONST robtarget Target_12860:=[[161.713599412,104.916728514,0],[0,0,1,0],[0,0,0,0],[9E+09,9E+09,9E+09,9E+09,9E+09,9E+09]];
    CONST robtarget Target_12870:=[[156.089396776,101.898276909,0],[0,0,1,0],[0,0,0,0],[9E+09,9E+09,9E+09,9E+09,9E+09,9E+09]];
    CONST robtarget Target_12880:=[[150.787771402,98.398834093,0],[0,0,1,0],[0,0,0,0],[9E+09,9E+09,9E+09,9E+09,9E+09,9E+09]];
    CONST robtarget Target_12890:=[[145.794660602,94.388936972,0],[0,0,1,0],[0,0,0,0],[9E+09,9E+09,9E+09,9E+09,9E+09,9E+09]];
    CONST robtarget Target_12900:=[[147.845449762,92.815849156,0],[0,0,1,0],[0,0,0,0],[9E+09,9E+09,9E+09,9E+09,9E+09,9E+09]];
    CONST robtarget Target_12910:=[[145.815759153,92.311765603,0],[0,0,1,0],[0,0,0,0],[9E+09,9E+09,9E+09,9E+09,9E+09,9E+09]];
    CONST robtarget Target_12920:=[[143.928526351,91.643121546,0],[0,0,1,0],[0,0,0,0],[9E+09,9E+09,9E+09,9E+09,9E+09,9E+09]];
    CONST robtarget Target_12930:=[[140.535895227,89.860328986,0],[0,0,1,0],[0,0,0,0],[9E+09,9E+09,9E+09,9E+09,9E+09,9E+09]];
    CONST robtarget Target_12940:=[[137.576478509,87.563825609,0],[0,0,1,0],[0,0,0,0],[9E+09,9E+09,9E+09,9E+09,9E+09,9E+09]];
    CONST robtarget Target_12950:=[[134.959198313,84.849965548,0],[0,0,1,0],[0,0,0,0],[9E+09,9E+09,9E+09,9E+09,9E+09,9E+09]];
    CONST robtarget Target_12960:=[[133.026641289,81.962755475,0],[0,0,1,0],[0,0,0,0],[9E+09,9E+09,9E+09,9E+09,9E+09,9E+09]];
    CONST robtarget Target_12970:=[[131.241018834,78.93836344,0],[0,0,1,0],[0,0,0,0],[9E+09,9E+09,9E+09,9E+09,9E+09,9E+09]];
    CONST robtarget Target_12980:=[[128.848526066,75.550363342,0],[0,0,1,0],[0,0,0,0],[9E+09,9E+09,9E+09,9E+09,9E+09,9E+09]];
    CONST robtarget Target_12990:=[[126.318917502,72.330238046,0],[0,0,1,0],[0,0,0,0],[9E+09,9E+09,9E+09,9E+09,9E+09,9E+09]];
    CONST robtarget Target_13000:=[[123.622809715,69.309677676,0],[0,0,1,0],[0,0,0,0],[9E+09,9E+09,9E+09,9E+09,9E+09,9E+09]];
    CONST robtarget Target_13010:=[[120.730819274,66.520372352,0],[0,0,1,0],[0,0,0,0],[9E+09,9E+09,9E+09,9E+09,9E+09,9E+09]];
    CONST robtarget Target_13020:=[[117.61356275,63.994012198,0],[0,0,1,0],[0,0,0,0],[9E+09,9E+09,9E+09,9E+09,9E+09,9E+09]];
    CONST robtarget Target_13030:=[[114.241656715,61.762287336,0],[0,0,1,0],[0,0,0,0],[9E+09,9E+09,9E+09,9E+09,9E+09,9E+09]];
    CONST robtarget Target_13040:=[[110.585717737,59.856887887,0],[0,0,1,0],[0,0,0,0],[9E+09,9E+09,9E+09,9E+09,9E+09,9E+09]];
    CONST robtarget Target_13050:=[[106.616362389,58.309503974,0],[0,0,1,0],[0,0,0,0],[9E+09,9E+09,9E+09,9E+09,9E+09,9E+09]];
    CONST robtarget Target_13060:=[[104.380938947,57.611993631,0],[0,0,1,0],[0,0,0,0],[9E+09,9E+09,9E+09,9E+09,9E+09,9E+09]];
    CONST robtarget Target_13070:=[[102.123990926,57.177040664,0],[0,0,1,0],[0,0,0,0],[9E+09,9E+09,9E+09,9E+09,9E+09,9E+09]];
    CONST robtarget Target_13080:=[[99.699786342,57.252076786,0],[0,0,1,0],[0,0,0,0],[9E+09,9E+09,9E+09,9E+09,9E+09,9E+09]];
    CONST robtarget Target_13090:=[[98.379421594,57.558163166,0],[0,0,1,0],[0,0,0,0],[9E+09,9E+09,9E+09,9E+09,9E+09,9E+09]];
    CONST robtarget Target_13100:=[[96.962593212,58.08453371,0],[0,0,1,0],[0,0,0,0],[9E+09,9E+09,9E+09,9E+09,9E+09,9E+09]];
    CONST robtarget Target_13110:=[[102.01949639,60.637305124,0],[0,0,1,0],[0,0,0,0],[9E+09,9E+09,9E+09,9E+09,9E+09,9E+09]];
    CONST robtarget Target_13120:=[[106.720449641,63.518372446,0],[0,0,1,0],[0,0,0,0],[9E+09,9E+09,9E+09,9E+09,9E+09,9E+09]];
    CONST robtarget Target_13130:=[[111.108762819,66.689360624,0],[0,0,1,0],[0,0,0,0],[9E+09,9E+09,9E+09,9E+09,9E+09,9E+09]];
    CONST robtarget Target_13140:=[[115.227745777,70.111894603,0],[0,0,1,0],[0,0,0,0],[9E+09,9E+09,9E+09,9E+09,9E+09,9E+09]];
    CONST robtarget Target_13150:=[[119.120708369,73.747599331,0],[0,0,1,0],[0,0,0,0],[9E+09,9E+09,9E+09,9E+09,9E+09,9E+09]];
    CONST robtarget Target_13160:=[[122.83096045,77.558099755,0],[0,0,1,0],[0,0,0,0],[9E+09,9E+09,9E+09,9E+09,9E+09,9E+09]];
    CONST robtarget Target_13170:=[[129.876572493,85.549987473,0],[0,0,1,0],[0,0,0,0],[9E+09,9E+09,9E+09,9E+09,9E+09,9E+09]];
    CONST robtarget Target_13170_2:=[[129.876572493,85.549987473,20],[0,0,1,0],[0,0,0,0],[9E+09,9E+09,9E+09,9E+09,9E+09,9E+09]];


    !***********************************************************
    !
    ! Module:  Module1
    !
    ! Description:
    !   <This program gives the user four options to choose from.
    !    1. The first option draw's the intials of the Author
    !    2. The second option draws a wolf. >
    !    3. The third lets the user start writing text on the flexpendant which then, is written down on the piece of paper.
    !    4. The last option is on the far left which lets the user decide the starting location and writes the text
    !
    !       (Note: this program only works with small letters and a few other characters)
    !
    ! Author: Raj
    !
    ! Version: 1.0
    !
    !***********************************************************

    !Error Message variables
    CONST errstr not_defined := "Not defined";
    CONST errstr not_defined_str1 := "The letter haas not been defined in this program.";

    !Main Program
    PROC main()

        !Default Values
        VAR num starting_x := 10;
        VAR num starting_y := 10;
        VAR num starting_z := 0;
        VAR num scaling := 3;
        VAR string text := "hello world";
        reg2 := 4;

        TPReadFK reg1, "What should the robot do?", "Manual write", stEmpty, "Draw Initials", "Draw wolf", "Write text";                        !Ask's which option the user would like to select and then goes to the appropriate option
        IF reg1 = 1 THEN                                                                                                                        !Lets the user decide the starting location for writing text and then write the text
            TPReadNum reg2, "Enter starting position (x)";
            TPReadNum reg3, "Enter starting position (y)";
            TPReadNum reg4, "Enter your font size";
            text := UIAlphaEntry(\Header:= "Manual write",\Message:= "What would you like to write"\Icon:=iconInfo,\InitString:= "text");
            starting_x := reg2;
            starting_y := reg3;
            scaling := reg4;
            IF starting_y > 0 AND starting_y < 420 AND starting_x > 0 AND starting_x < 270 THEN                                                 !Check if the x and y location is inside the A3 sheet, if not give an error
                execute_command text, starting_x, starting_y, starting_z, scaling;
            ELSE
                ErrWrite "Location error", "Location is outside the A3 sheet" \RL2:="Start with a new A3 sheet";
                Stop;

            ENDIF
        ELSEIF reg1 = 3 THEN
            TPWrite "Writing Initials";                                                                                                         !Starts to write the author's initials
            Initials;
        ELSEIF reg1 = 4 THEN
            TPWrite "Starting to draw Wolf";                                                                                                    !Goes through the paths that were auto generated by using the AutoPath option in RobotStudio
            Wolf_Outline;
            Wolf_Upper;
            Wolf_Upper_2;
            Wolf_Mid;
            Wolf_Lower;
            Wolf_Paw;
            Wolf_Paw_2;
            Wolf_Paw_3;
            Wolf_Lower_2;
            Wolf_Outline_2;
        ELSEIF reg1 = 5 THEN                                                                                                                    !Let's the user write text starting from the top right corner
            TPReadNum reg4, "Enter your font size";

            ! Calculating the starting position depending on the font size
            scaling := reg4;
            starting_x := 10 + .5 * scaling;
            starting_y := 390 - scaling * scaling * scaling;

            !Wait for the user to write text and then keep on running until the user wants to stop writing
            WHILE reg2 <= 4 DO
                TPReadFK reg2, "What should the robot do?", "Font size", stEmpty, stEmpty, "Write", "Finish writing";
                IF reg2 = 4 THEN
                text := UIAlphaEntry(\Header:= "Write text",\Message:= "Write your text below?"\Icon:=iconInfo,\InitString:= "an example");

            !Checks if there is space in the A3 sheet, if not stops the programe and gives an error message
                    IF starting_y > 0 THEN
                        execute_command text, starting_x, starting_y, starting_z, scaling;
                        starting_y := update_pos_y(text, starting_y,scaling);
                    ELSE
                        ErrWrite "Location error", "Location is outside the A3 sheet" \RL2:="Start with a new A3 sheet";
                        Stop;
                    ENDIF
                ELSEIF reg2 = 1 THEN
                    TPReadNum reg4, "Enter your font size";
                    scaling := reg4;
                    starting_y := starting_y - 8 *scaling;
                ENDIF

            ENDWHILE
        ENDIF
    ENDPROC


    FUNC num update_pos_y(string text, num y, num scaling)                                                                                      !checks the length of the string AND decide how many lines have been written, then updates the new y value
        VAR num new_y;
        VAR num lines;

        IF (10 + .5 * scaling + strlen(text)*scaling*6 + 9 * scaling) > (297 - 10 - 6 * scaling) THEN
            lines := (10 + .5 * scaling + strlen(text)*scaling*6+ 9 * scaling)/(297 - 10 - 6 * scaling);
            IF lines - round(lines) >= 0 THEN
                lines := round(lines) + 1;
            ELSE
                lines := round(lines);
            ENDIF
            new_y := y - 17 * scaling * lines;
        ELSE
            new_y := y - 17 * scaling;
        ENDIF
        RETURN new_y;
    ENDFUNC

   PROC execute_command(string text, num x, num y, num z, num scaling)                                                                          !Decide the x and y location for each letter and one by one send the letter to a procedure that decides what letter to write

        VAR num string_length;
        VAR string current_string;
        string_length:= strlen(text);

        !Start going through each letter
        FOR I FROM 1 to string_length STEP + 1 DO
            IF I = 1 THEN
                TPWrite "Starting to write";
            ENDIF
        current_string := StrPart(text,I,1);

        !Check if the robot taget is within the x axis of the A3 sheet, if not set a new x and y position
        IF current_string = "i" OR current_string = "l" OR current_string = " " OR current_string = "." THEN
            IF x >= 297 - 10 - 4 * scaling THEN
                dash x, y, z, scaling;
                y := y - 15 * scaling;
                x := 10 + .5 * scaling;
            ENDIF
        ELSEIF current_string = "f" OR current_string = "t" OR current_string = "j" THEN
            IF x >= 297 - 10 - 6 * scaling THEN
                dash x, y, z, scaling;
                y := y - 15 * scaling;
                x := 10 + .5 * scaling;
            ENDIF
        ELSEIF current_string = "m" OR current_string = "w" THEN
            IF x >= 297 - 10 - 12 * scaling THEN
                dash x, y, z, scaling;
                y := y - 15 * scaling;
                x := 10 + .5 * scaling;
            ENDIF
        ELSEIF x >= 297 - 10 - 6 * scaling THEN
            dash x, y, z, scaling;
            y := y - 15 * scaling;
            x := 10 + .5 * scaling;
        ENDIF

        !Wrtite the current letter
        IF y > 0 THEN
            write_letter current_string, x, y, z, scaling;
        ELSE
            ErrWrite "Location error", "Location is outside the A3 sheet" \RL2:="Start with a new A3 sheet";
            Stop;
        ENDIF


        !Update the x and y after writing the letter
        IF current_string = "i" OR current_string = "l" OR current_string = " " OR current_string = "." THEN
            IF current_string = " " THEN
                x := x + 2 * scaling*2;
            ELSE
                x := x + 2 * scaling;
            ENDIF
        ELSEIF current_string = "f" OR current_string = "t" OR current_string = "j" THEN
            x := x + 6 * scaling;
        ELSEIF current_string = "m" OR current_string = "w" THEN
            x := x + 14 * scaling;
        ELSE
            x := x + 8 * scaling;
        ENDIF
        ENDFOR

   ENDPROC

    PROC write_letter(string letter,num x, num y,num z, num scaling)                                                                            !Check which letter it is and then go to the right procedure, if the letter or character has not been defined give an error message
        IF letter = "a" THEN
            a x, y, z, scaling;
        ELSEIF letter = "b" THEN
            b x, y, z, scaling;
        ELSEIF letter = "c" THEN
            c x, y, z, scaling;
        ELSEIF letter = "d" THEN
            d x, y, z, scaling;
        ELSEIF letter = "e" THEN
            e x, y, z, scaling;
        ELSEIF letter = "f" THEN
            f x, y, z, scaling;
        ELSEIF letter = "g" THEN
            g x, y, z, scaling;
        ELSEIF letter = "h" THEN
            h x, y, z, scaling;
        ELSEIF letter = "i" THEN
            i x, y, z, scaling;
        ELSEIF letter = "j" THEN
            j x, y, z, scaling;
        ELSEIF letter = "k" THEN
            k x, y, z, scaling;
        ELSEIF letter = "l" THEN
            l x, y, z, scaling;
        ELSEIF letter = "m" THEN
            m x, y, z, scaling;
        ELSEIF letter = "n" THEN
            n x, y, z, scaling;
        ELSEIF letter = "o" THEN
            o x, y, z, scaling;
        ELSEIF letter = "p" THEN
            p x, y, z, scaling;
        ELSEIF letter = "q" THEN
            q x, y, z, scaling;
        ELSEIF letter = "r" THEN
            r x, y, z, scaling;
        ELSEIF letter = "s" THEN
            s x, y, z, scaling;
        ELSEIF letter = "t" THEN
            t x, y, z, scaling;
        ELSEIF letter = "u" THEN
            u x, y, z, scaling;
        ELSEIF letter = "v" THEN
            v x, y, z, scaling;
        ELSEIF letter = "w" THEN
            w x, y, z, scaling;
        ELSEIF letter = "x" THEN
            x_draw x, y, z, scaling;
        ELSEIF letter = "y" THEN
            y_draw x, y, z, scaling;
        ELSEIF letter = "z" THEN
            z_draw x, y, z, scaling;
        ELSEIF letter = "-" THEN
            dash x, y, z, scaling;
        ELSEIF letter = "." THEN
            dot x, y, z, scaling;
        ELSEIF letter = "?" THEN
            question x, y, z, scaling;
        ELSEIF letter = " " THEN
            !pass
        ELSE
            ErrLog 4800 , not_defined, not_defined_str1, ERRSTR_EMPTY, ERRSTR_EMPTY,ERRSTR_UNUSED;
            WaitTime 6;

        ENDIF
    ENDPROC

!Below are the defined targets to write each individual letter and some other characters
	PROC a(num starting_x, num starting_y, num starting_z, num scaling)
        VAR robtarget a_0;
        VAR robtarget a_1;
        VAR robtarget a_2;
	    VAR robtarget a_3;
	    VAR robtarget a_4;
	    VAR robtarget a_5;
	    VAR robtarget a_6;
	    VAR robtarget a_7;
	    VAR robtarget a_8;
	    VAR robtarget a_9;
	    VAR robtarget a_10;
	    VAR robtarget a_11;
	    VAR robtarget a_12;
        VAR robtarget a_13;

        a_0:=[[starting_x + 0.5 * scaling, starting_y + 8 * scaling, starting_z + 20],[0,0,1,0],[0,0,0,0],[9E+09,9E+09,9E+09,9E+09,9E+09,9E+09]];
        a_1:=[[starting_x + 0.5 * scaling, starting_y + 8 * scaling, starting_z + 0],[0,0,1,0],[0,0,0,0],[9E+09,9E+09,9E+09,9E+09,9E+09,9E+09]];
        a_2:=[[starting_x + 3.5 * scaling, starting_y + 9 * scaling, starting_z + 0],[0,0,1,0],[0,0,0,0],[9E+09,9E+09,9E+09,9E+09,9E+09,9E+09]];
        a_3:=[[starting_x + 6 * scaling, starting_y + 8 * scaling, starting_z + 0],[0,0,1,0],[0,0,0,0],[9E+09,9E+09,9E+09,9E+09,9E+09,9E+09]];
        a_4:=[[starting_x + 6.35 * scaling, starting_y + 7 * scaling, starting_z + 0],[0,0,1,0],[0,0,0,0],[9E+09,9E+09,9E+09,9E+09,9E+09,9E+09]];
        a_5:=[[starting_x + 6.5 * scaling, starting_y + 6 * scaling, starting_z + 0],[0,0,1,0],[0,0,0,0],[9E+09,9E+09,9E+09,9E+09,9E+09,9E+09]];
        a_6:=[[starting_x + 6.5 * scaling, starting_y + 0 * scaling, starting_z + 0],[0,0,1,0],[0,0,0,0],[9E+09,9E+09,9E+09,9E+09,9E+09,9E+09]];
        a_7:=[[starting_x + 6.5 * scaling, starting_y + 1.3 * scaling, starting_z + 0],[0,0,1,0],[0,0,0,0],[9E+09,9E+09,9E+09,9E+09,9E+09,9E+09]];
        a_8:=[[starting_x + 3.5 * scaling, starting_y + 0 * scaling, starting_z + 0],[0,0,1,0],[0,0,0,0],[9E+09,9E+09,9E+09,9E+09,9E+09,9E+09]];
        a_9:=[[starting_x + 0 * scaling, starting_y + 2.5 * scaling, starting_z + 0],[0,0,1,0],[0,0,0,0],[9E+09,9E+09,9E+09,9E+09,9E+09,9E+09]];
        a_10:=[[starting_x + 1 * scaling, starting_y + 4.5 * scaling, starting_z + 0],[0,0,1,0],[0,0,0,0],[9E+09,9E+09,9E+09,9E+09,9E+09,9E+09]];
        a_11:=[[starting_x + 3 * scaling,starting_y + 5 * scaling, starting_z + 0],[0,0,1,0],[0,0,0,0],[9E+09,9E+09,9E+09,9E+09,9E+09,9E+09]];
        a_12:=[[starting_x + 6.5 * scaling,starting_y + 5 * scaling, starting_z + 0],[0,0,1,0],[0,0,0,0],[9E+09,9E+09,9E+09,9E+09,9E+09,9E+09]];
        a_13:=[[starting_x + 6.5 * scaling,starting_y + 5 * scaling, starting_z + 20],[0,0,1,0],[0,0,0,0],[9E+09,9E+09,9E+09,9E+09,9E+09,9E+09]];

        MoveL a_0,v50,fine,MyNewTool\WObj:=A3;
	    MoveL a_1,v50,fine,MyNewTool\WObj:=A3;
	    MoveC a_2,a_3,v50,fine,MyNewTool\WObj:=A3;
	    MoveC a_4,a_5,v50,fine,MyNewTool\WObj:=A3;
	    MoveL a_6,v50,fine,MyNewTool\WObj:=A3;
	    MoveL a_7,v50,fine,MyNewTool\WObj:=A3;
	    MoveC a_8,a_9,v50,z5,MyNewTool\WObj:=A3;
	    MoveC a_10,a_11,v50,fine,MyNewTool\WObj:=A3;
	    MoveL a_12,v50,fine,MyNewTool\WObj:=A3;
        MoveL a_13,v50,fine,MyNewTool\WObj:=A3;

	ENDPROC

    PROC b(num starting_x, num starting_y, num starting_z, num scaling)
        VAR robtarget b_0;
        VAR robtarget b_1;
        VAR robtarget b_2;
	    VAR robtarget b_3;
	    VAR robtarget b_4;
	    VAR robtarget b_5;
	    VAR robtarget b_6;
	    VAR robtarget b_7;
	    VAR robtarget b_8;
	    VAR robtarget b_9;
	    VAR robtarget b_10;

        b_0:=[[starting_x + 0 * scaling, starting_y + 14 * scaling, starting_z + 20],[0,0,1,0],[0,0,0,0],[9E+09,9E+09,9E+09,9E+09,9E+09,9E+09]];
        b_1:=[[starting_x + 0 * scaling, starting_y + 14 * scaling, starting_z + 0],[0,0,1,0],[0,0,0,0],[9E+09,9E+09,9E+09,9E+09,9E+09,9E+09]];
        b_2:=[[starting_x + 0 * scaling, starting_y + 0 * scaling, starting_z + 0],[0,0,1,0],[0,0,0,0],[9E+09,9E+09,9E+09,9E+09,9E+09,9E+09]];
        b_3:=[[starting_x + 0 * scaling, starting_y + 2 * scaling, starting_z + 0],[0,0,1,0],[0,0,0,0],[9E+09,9E+09,9E+09,9E+09,9E+09,9E+09]];
        b_4:=[[starting_x + 3.5 * scaling, starting_y + 0 * scaling, starting_z + 0],[0,0,1,0],[0,0,0,0],[9E+09,9E+09,9E+09,9E+09,9E+09,9E+09]];
        b_5:=[[starting_x + 6 * scaling, starting_y + 2 * scaling, starting_z + 0],[0,0,1,0],[0,0,0,0],[9E+09,9E+09,9E+09,9E+09,9E+09,9E+09]];
        b_6:=[[starting_x + 6.5 * scaling, starting_y + 5 * scaling, starting_z + 0],[0,0,1,0],[0,0,0,0],[9E+09,9E+09,9E+09,9E+09,9E+09,9E+09]];
        b_7:=[[starting_x + 5.5 * scaling, starting_y + 8 * scaling, starting_z + 0],[0,0,1,0],[0,0,0,0],[9E+09,9E+09,9E+09,9E+09,9E+09,9E+09]];
        b_8:=[[starting_x + 3 * scaling, starting_y + 9 * scaling, starting_z + 0],[0,0,1,0],[0,0,0,0],[9E+09,9E+09,9E+09,9E+09,9E+09,9E+09]];
        b_9:=[[starting_x + 0 * scaling, starting_y + 7 * scaling, starting_z + 0],[0,0,1,0],[0,0,0,0],[9E+09,9E+09,9E+09,9E+09,9E+09,9E+09]];
        b_10:=[[starting_x + 0 * scaling, starting_y + 7 * scaling, starting_z + 20],[0,0,1,0],[0,0,0,0],[9E+09,9E+09,9E+09,9E+09,9E+09,9E+09]];

        MoveL b_0,v50,fine,MyNewTool\WObj:=A3;
	    MoveL b_1,v50,fine,MyNewTool\WObj:=A3;
        MoveL b_2,v50,fine,MyNewTool\WObj:=A3;
        MoveL b_3,v50,fine,MyNewTool\WObj:=A3;
	    MoveC b_4,b_5,v50,fine,MyNewTool\WObj:=A3;
	    MoveC b_6,b_7,v50,fine,MyNewTool\WObj:=A3;
	    MoveC b_8,b_9,v50,fine,MyNewTool\WObj:=A3;
	    MoveL b_10,v50,fine,MyNewTool\WObj:=A3;

	ENDPROC

    PROC c(num starting_x, num starting_y, num starting_z, num scaling)
        VAR robtarget c_0;
        VAR robtarget c_1;
        VAR robtarget c_2;
	    VAR robtarget c_3;
	    VAR robtarget c_4;
	    VAR robtarget c_5;
	    VAR robtarget c_6;

        c_0:=[[starting_x + 6 * scaling, starting_y + 8 * scaling, starting_z + 20],[0,0,1,0],[0,0,0,0],[9E+09,9E+09,9E+09,9E+09,9E+09,9E+09]];
        c_1:=[[starting_x + 6 * scaling, starting_y + 8 * scaling, starting_z + 0],[0,0,1,0],[0,0,0,0],[9E+09,9E+09,9E+09,9E+09,9E+09,9E+09]];
        c_2:=[[starting_x + 3 * scaling, starting_y + 9 * scaling, starting_z + 0],[0,0,1,0],[0,0,0,0],[9E+09,9E+09,9E+09,9E+09,9E+09,9E+09]];
        c_3:=[[starting_x + 0 * scaling, starting_y + 5 * scaling, starting_z + 0],[0,0,1,0],[0,0,0,0],[9E+09,9E+09,9E+09,9E+09,9E+09,9E+09]];
        c_4:=[[starting_x + 3 * scaling, starting_y + 0.5 * scaling, starting_z + 0],[0,0,1,0],[0,0,0,0],[9E+09,9E+09,9E+09,9E+09,9E+09,9E+09]];
        c_5:=[[starting_x + 6 * scaling, starting_y + 1 * scaling, starting_z + 0],[0,0,1,0],[0,0,0,0],[9E+09,9E+09,9E+09,9E+09,9E+09,9E+09]];
        c_6:=[[starting_x + 6 * scaling, starting_y + 1 * scaling, starting_z + 20],[0,0,1,0],[0,0,0,0],[9E+09,9E+09,9E+09,9E+09,9E+09,9E+09]];


        MoveL c_0,v50,fine,MyNewTool\WObj:=A3;
        MoveL c_1,v50,fine,MyNewTool\WObj:=A3;
	    MoveC c_2,c_3,v50,z5,MyNewTool\WObj:=A3;
	    MoveC c_4,c_5,v50,fine,MyNewTool\WObj:=A3;
	    MoveL c_6,v50,fine,MyNewTool\WObj:=A3;

    ENDPROC

    PROC d(num starting_x, num starting_y, num starting_z, num scaling)
        VAR robtarget d_0;
        VAR robtarget d_1;
        VAR robtarget d_2;
	    VAR robtarget d_3;
	    VAR robtarget d_4;
	    VAR robtarget d_5;
	    VAR robtarget d_6;
	    VAR robtarget d_7;
	    VAR robtarget d_8;
	    VAR robtarget d_9;
	    VAR robtarget d_10;

        d_0:=[[starting_x + 6.5* scaling, starting_y + 14 * scaling, starting_z + 20],[0,0,1,0],[0,0,0,0],[9E+09,9E+09,9E+09,9E+09,9E+09,9E+09]];
        d_1:=[[starting_x + 6.5 * scaling, starting_y + 14 * scaling, starting_z + 0],[0,0,1,0],[0,0,0,0],[9E+09,9E+09,9E+09,9E+09,9E+09,9E+09]];
        d_2:=[[starting_x + 6.5 * scaling, starting_y + 0 * scaling, starting_z + 0],[0,0,1,0],[0,0,0,0],[9E+09,9E+09,9E+09,9E+09,9E+09,9E+09]];
        d_3:=[[starting_x + 6.5 * scaling, starting_y + 2 * scaling, starting_z + 0],[0,0,1,0],[0,0,0,0],[9E+09,9E+09,9E+09,9E+09,9E+09,9E+09]];
        d_4:=[[starting_x + 3.5 * scaling, starting_y + 0 * scaling, starting_z + 0],[0,0,1,0],[0,0,0,0],[9E+09,9E+09,9E+09,9E+09,9E+09,9E+09]];
        d_5:=[[starting_x + 0.5 * scaling, starting_y + 2 * scaling, starting_z + 0],[0,0,1,0],[0,0,0,0],[9E+09,9E+09,9E+09,9E+09,9E+09,9E+09]];
        d_6:=[[starting_x + 0 * scaling, starting_y + 5 * scaling, starting_z + 0],[0,0,1,0],[0,0,0,0],[9E+09,9E+09,9E+09,9E+09,9E+09,9E+09]];
        d_7:=[[starting_x + 1.2 * scaling, starting_y + 8 * scaling, starting_z + 0],[0,0,1,0],[0,0,0,0],[9E+09,9E+09,9E+09,9E+09,9E+09,9E+09]];
        d_8:=[[starting_x + 3.5 * scaling, starting_y + 9 * scaling, starting_z + 0],[0,0,1,0],[0,0,0,0],[9E+09,9E+09,9E+09,9E+09,9E+09,9E+09]];
        d_9:=[[starting_x + 6.5 * scaling, starting_y + 7 * scaling, starting_z + 0],[0,0,1,0],[0,0,0,0],[9E+09,9E+09,9E+09,9E+09,9E+09,9E+09]];
        d_10:=[[starting_x + 6.5 * scaling, starting_y + 7 * scaling, starting_z + 20],[0,0,1,0],[0,0,0,0],[9E+09,9E+09,9E+09,9E+09,9E+09,9E+09]];

        MoveL d_0,v50,fine,MyNewTool\WObj:=A3;
	    MoveL d_1,v50,fine,MyNewTool\WObj:=A3;
        MoveL d_2,v50,fine,MyNewTool\WObj:=A3;
        MoveL d_3,v50,fine,MyNewTool\WObj:=A3;
	    MoveC d_4,d_5,v50,fine,MyNewTool\WObj:=A3;
	    MoveC d_6,d_7,v50,fine,MyNewTool\WObj:=A3;
	    MoveC d_8,d_9,v50,fine,MyNewTool\WObj:=A3;
	    MoveL d_10,v50,fine,MyNewTool\WObj:=A3;

	ENDPROC

     PROC e(num starting_x, num starting_y,  num starting_z, num scaling)
        VAR robtarget e_0;
        VAR robtarget e_1;
        VAR robtarget e_2;
	    VAR robtarget e_3;
	    VAR robtarget e_4;
	    VAR robtarget e_5;
	    VAR robtarget e_6;
        VAR robtarget e_7;
        VAR robtarget e_8;
        VAR robtarget e_9;

        e_0:=[[starting_x + 7 * scaling, starting_y + 1 * scaling, starting_z + 20],[0,0,1,0],[0,0,0,0],[9E+09,9E+09,9E+09,9E+09,9E+09,9E+09]];
        e_1:=[[starting_x + 7 * scaling, starting_y + 1 * scaling, starting_z + 0],[0,0,1,0],[0,0,0,0],[9E+09,9E+09,9E+09,9E+09,9E+09,9E+09]];
        e_2:=[[starting_x + 4 * scaling, starting_y + 0 * scaling, starting_z + 0],[0,0,1,0],[0,0,0,0],[9E+09,9E+09,9E+09,9E+09,9E+09,9E+09]];
        e_3:=[[starting_x + 1 * scaling, starting_y + 1 * scaling, starting_z + 0],[0,0,1,0],[0,0,0,0],[9E+09,9E+09,9E+09,9E+09,9E+09,9E+09]];
        e_4:=[[starting_x + 0 * scaling, starting_y + 5 * scaling, starting_z + 0],[0,0,1,0],[0,0,0,0],[9E+09,9E+09,9E+09,9E+09,9E+09,9E+09]];
        e_5:=[[starting_x + 1 * scaling, starting_y + 8 * scaling, starting_z + 0],[0,0,1,0],[0,0,0,0],[9E+09,9E+09,9E+09,9E+09,9E+09,9E+09]];
        e_6:=[[starting_x + 5.5 * scaling, starting_y + 9 * scaling, starting_z + 0],[0,0,1,0],[0,0,0,0],[9E+09,9E+09,9E+09,9E+09,9E+09,9E+09]];
        e_7:=[[starting_x + 7 * scaling, starting_y + 5 * scaling, starting_z + 0],[0,0,1,0],[0,0,0,0],[9E+09,9E+09,9E+09,9E+09,9E+09,9E+09]];
        e_8:=[[starting_x + 0 * scaling, starting_y + 5 * scaling, starting_z + 0],[0,0,1,0],[0,0,0,0],[9E+09,9E+09,9E+09,9E+09,9E+09,9E+09]];
        e_9:=[[starting_x + 0 * scaling, starting_y + 5 * scaling, starting_z + 20],[0,0,1,0],[0,0,0,0],[9E+09,9E+09,9E+09,9E+09,9E+09,9E+09]];

        MoveL e_0,v50,fine,MyNewTool\WObj:=A3;
        MoveL e_1,v50,fine,MyNewTool\WObj:=A3;
        MoveC e_2,e_3,v50,z5,MyNewTool\WObj:=A3;
	    MoveC e_4,e_5,v50,z1,MyNewTool\WObj:=A3;
        MoveC e_6,e_7,v50,z1,MyNewTool\WObj:=A3;
	    MoveL e_8,v50,fine,MyNewTool\WObj:=A3;
        MoveL e_9,v50,fine,MyNewTool\WObj:=A3;

    ENDPROC

    PROC f(num starting_x, num starting_y, num starting_z, num scaling)
        VAR robtarget f_0;
        VAR robtarget f_1;
        VAR robtarget f_2;
	    VAR robtarget f_3;
	    VAR robtarget f_4;
	    VAR robtarget f_5;
	    VAR robtarget f_6;
        VAR robtarget f_7;
        VAR robtarget f_8;
        VAR robtarget f_9;

        f_0:=[[starting_x + 2 * scaling, starting_y + 0 * scaling, starting_z + 20],[0,0,1,0],[0,0,0,0],[9E+09,9E+09,9E+09,9E+09,9E+09,9E+09]];
        f_1:=[[starting_x + 2 * scaling, starting_y + 0 * scaling, starting_z + 0],[0,0,1,0],[0,0,0,0],[9E+09,9E+09,9E+09,9E+09,9E+09,9E+09]];
        f_2:=[[starting_x + 2 * scaling, starting_y + 11 * scaling, starting_z + 0],[0,0,1,0],[0,0,0,0],[9E+09,9E+09,9E+09,9E+09,9E+09,9E+09]];
        f_3:=[[starting_x + 3 * scaling, starting_y + 13 * scaling, starting_z + 0],[0,0,1,0],[0,0,0,0],[9E+09,9E+09,9E+09,9E+09,9E+09,9E+09]];
        f_4:=[[starting_x + 5.5 * scaling, starting_y + 13 * scaling, starting_z + 0],[0,0,1,0],[0,0,0,0],[9E+09,9E+09,9E+09,9E+09,9E+09,9E+09]];
        f_5:=[[starting_x + 5.5 * scaling, starting_y + 13 * scaling, starting_z + 20],[0,0,1,0],[0,0,0,0],[9E+09,9E+09,9E+09,9E+09,9E+09,9E+09]];
        f_6:=[[starting_x + 0 * scaling, starting_y + 9 * scaling, starting_z + 20],[0,0,1,0],[0,0,0,0],[9E+09,9E+09,9E+09,9E+09,9E+09,9E+09]];
        f_7:=[[starting_x + 0 * scaling, starting_y + 9 * scaling, starting_z + 0],[0,0,1,0],[0,0,0,0],[9E+09,9E+09,9E+09,9E+09,9E+09,9E+09]];
        f_8:=[[starting_x + 5 * scaling, starting_y + 9 * scaling, starting_z + 0],[0,0,1,0],[0,0,0,0],[9E+09,9E+09,9E+09,9E+09,9E+09,9E+09]];
        f_9:=[[starting_x + 5 * scaling, starting_y + 9 * scaling, starting_z + 20],[0,0,1,0],[0,0,0,0],[9E+09,9E+09,9E+09,9E+09,9E+09,9E+09]];

        MoveL f_0,v50,fine,MyNewTool\WObj:=A3;
        MoveL f_1,v50,fine,MyNewTool\WObj:=A3;
        MoveL f_2,v50,fine,MyNewTool\WObj:=A3;
	    MoveC f_3,f_4,v50,fine,MyNewTool\WObj:=A3;
        MoveL f_5,v50,fine,MyNewTool\WObj:=A3;
	    MoveL f_6,v50,fine,MyNewTool\WObj:=A3;
        MoveL f_7,v50,fine,MyNewTool\WObj:=A3;
        MoveL f_8,v50,fine,MyNewTool\WObj:=A3;
        MoveL f_9,v50,fine,MyNewTool\WObj:=A3;

    ENDPROC

    PROC g(num starting_x, num starting_y, num starting_z, num scaling)
        VAR robtarget g_0;
        VAR robtarget g_1;
        VAR robtarget g_2;
	    VAR robtarget g_3;
	    VAR robtarget g_4;
	    VAR robtarget g_5;
	    VAR robtarget g_6;
        VAR robtarget g_7;
        VAR robtarget g_8;
        VAR robtarget g_9;
        VAR robtarget g_10;
        VAR robtarget g_11;
        VAR robtarget g_12;
        VAR robtarget g_13;
        VAR robtarget g_14;
        VAR robtarget g_15;
        VAR robtarget g_16;
        VAR robtarget g_17;
        VAR robtarget g_18;
        VAR robtarget g_19;

